KUKA KRL program: MyProgram_188().src

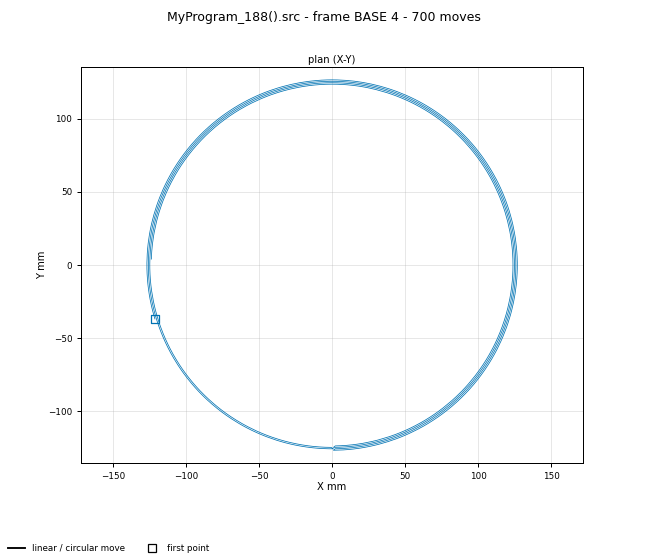
[picture p0: tool path of MyProgram_188().src in frame BASE 4, 700 of 700 moves have a stored position in this frame; points joined in program order, loops and branches not executed]
&ACCESS RVP
&REL 1
&PARAM TEMPLATE = C:\KRC\Roboter\Template\vorgabe
&PARAM EDITMASK = *
DEF MyProgram_188()
; ---- Setting reference (Base) ----
$BASE = BASE_DATA[4]

; --------------------------
; ---- Setting tool (TCP) ----
$TOOL = TOOL_DATA[3]
; --------------------------

$VEL.CP = VEL_APROX_PRINT
Startdeposition()
$VEL.CP = VEL_PRINT
LIN {X -121.2138,Y -36.8642,Z 137,A -166.8742,B 24.9598,C -1.4645,E1 24.8465,E2 613.2889} C_DIS
LIN {X -122.0831,Y -33.8748,Z 137,A -168.3082,B 24.9596,C -1.4677,E1 24.8454,E2 614.7236} C_DIS
LIN {X -122.8265,Y -31.0709,Z 137,A -169.6455,B 24.9595,C -1.4706,E1 24.8445,E2 616.0617} C_DIS
LIN {X -123.5708,Y -27.965,Z 137,A -171.133,B 24.9593,C -1.4732,E1 24.8435,E2 617.5517} C_DIS
LIN {X -124.4803,Y -23.589,Z 137,A -173.1147,B 24.9589,C -1.4814,E1 24.8424,E2 619.5256} C_DIS
LIN {X -125.0881,Y -20.1308,Z 137,A -174.7108,B 24.9586,C -1.4861,E1 24.8417,E2 621.1201} C_DIS
LIN {X -125.6254,Y -16.433,Z 137,A -176.4459,B 24.9584,C -1.4895,E1 24.841,E2 622.8573} C_DIS
LIN {X -126.0094,Y -13.1745,Z 137,A -177.8897,B 24.9581,C -1.4961,E1 24.8406,E2 624.2941} C_DIS
LIN {X -126.3219,Y -9.7379,Z 137,A -179.5918,B 24.9581,C -1.4948,E1 24.8402,E2 626.0096} C_DIS
LIN {X -126.5479,Y -6.1219,Z 137,A 178.8842,B 24.9575,C -1.5053,E1 24.8399,E2 627.5177} C_DIS
LIN {X -126.67,Y -2.6015,Z 137,A 177.1602,B 24.9575,C -1.5046,E1 24.8399,E2 629.2537} C_DIS
LIN {X -126.6899,Y 1.403,Z 137,A 175.4591,B 24.957,C -1.5155,E1 24.8399,E2 630.9392} C_DIS
LIN {X -126.5902,Y 5.1764,Z 137,A 173.7113,B 24.9568,C -1.5193,E1 24.8399,E2 632.6884} C_DIS
LIN {X -126.4456,Y 7.9589,Z 137,A 172.4536,B 24.9565,C -1.5235,E1 24.8402,E2 633.9435} C_DIS
LIN {X -126.1864,Y 11.3702,Z 137,A 170.907,B 24.9562,C -1.5286,E1 24.8405,E2 635.4873} C_DIS
LIN {X -125.7902,Y 15.1199,Z 137,A 169.1622,B 24.956,C -1.5325,E1 24.8411,E2 637.2334} C_DIS
LIN {X -125.3864,Y 18.1682,Z 137,A 167.7803,B 24.9557,C -1.5374,E1 24.8416,E2 638.6117} C_DIS
LIN {X -124.9317,Y 21.0685,Z 137,A 166.3962,B 24.9557,C -1.5392,E1 24.8422,E2 639.9998} C_DIS
LIN {X -124.3869,Y 24.0779,Z 137,A 165.0026,B 24.9554,C -1.5433,E1 24.8429,E2 641.392} C_DIS
LIN {X -123.5065,Y 28.2467,Z 137,A 163.0731,B 24.955,C -1.5494,E1 24.8441,E2 643.3182} C_DIS
LIN {X -122.739,Y 31.4153,Z 137,A 161.63,B 24.9547,C -1.5556,E1 24.845,E2 644.7551} C_DIS
LIN {X -121.9722,Y 34.2715,Z 137,A 160.2417,B 24.9545,C -1.5576,E1 24.8461,E2 646.1466} C_DIS
LIN {X -120.9226,Y 37.8158,Z 137,A 158.5823,B 24.9542,C -1.5635,E1 24.8474,E2 647.8016} C_DIS
LIN {X -120.1284,Y 40.2607,Z 137,A 157.4077,B 24.954,C -1.5666,E1 24.8484,E2 648.9753} C_DIS
LIN {X -119.0964,Y 43.2181,Z 137,A 155.982,B 24.9538,C -1.5707,E1 24.8498,E2 650.3994} C_DIS
LIN {X -117.9044,Y 46.3735,Z 137,A 154.4616,B 24.9535,C -1.5757,E1 24.8513,E2 651.9164} C_DIS
LIN {X -116.6051,Y 49.5537,Z 137,A 152.8791,B 24.9533,C -1.5792,E1 24.853,E2 653.4993} C_DIS
LIN {X -115.5382,Y 51.9875,Z 137,A 151.6701,B 24.9531,C -1.5826,E1 24.8543,E2 654.7069} C_DIS
LIN {X -114.1439,Y 54.9818,Z 137,A 150.1755,B 24.9528,C -1.5871,E1 24.8561,E2 656.1989} C_DIS
LIN {X -112.5436,Y 58.1916,Z 137,A 148.4062,B 24.9529,C -1.5853,E1 24.8584,E2 657.9819} C_DIS
LIN {X -110.5519,Y 61.8908,Z 137,A 146.5051,B 24.9526,C -1.591,E1 24.8609,E2 659.8796} C_DIS
LIN {X -108.3456,Y 65.6764,Z 137,A 144.5451,B 24.9522,C -1.5977,E1 24.8637,E2 661.8337} C_DIS
LIN {X -106.0689,Y 69.2941,Z 137,A 142.5626,B 24.952,C -1.601,E1 24.8667,E2 663.8183} C_DIS
LIN {X -103.768,Y 72.6946,Z 137,A 140.68,B 24.9517,C -1.6051,E1 24.8697,E2 665.7005} C_DIS
LIN {X -101.3771,Y 75.9934,Z 137,A 138.8143,B 24.9515,C -1.6091,E1 24.8728,E2 667.5656} C_DIS
LIN {X -98.705,Y 79.4322,Z 137,A 136.8715,B 24.9511,C -1.6156,E1 24.8761,E2 669.5021} C_DIS
LIN {X -95.9842,Y 82.6994,Z 137,A 134.9801,B 24.9507,C -1.6221,E1 24.8795,E2 671.3866} C_DIS
LIN {X -93.1998,Y 85.8252,Z 137,A 133.087,B 24.9504,C -1.627,E1 24.8831,E2 673.2766} C_DIS
LIN {X -90.3574,Y 88.8127,Z 137,A 131.2166,B 24.9501,C -1.6314,E1 24.8867,E2 675.1446} C_DIS
LIN {X -87.5001,Y 91.629,Z 137,A 129.3359,B 24.9501,C -1.6328,E1 24.8905,E2 677.0299} C_DIS
LIN {X -84.2229,Y 94.651,Z 137,A 127.3353,B 24.9497,C -1.6382,E1 24.8946,E2 679.0256} C_DIS
LIN {X -81.1209,Y 97.3227,Z 137,A 125.4906,B 24.9494,C -1.6427,E1 24.8985,E2 680.8666} C_DIS
LIN {X -77.9388,Y 99.8892,Z 137,A 123.5646,B 24.9494,C -1.6432,E1 24.9027,E2 682.7985} C_DIS
LIN {X -74.6821,Y 102.3469,Z 137,A 121.7215,B 24.9492,C -1.6472,E1 24.9069,E2 684.6387} C_DIS
LIN {X -71.2136,Y 104.7894,Z 137,A 119.7906,B 24.9489,C -1.6506,E1 24.9113,E2 686.5683} C_DIS
LIN {X -67.4012,Y 107.2814,Z 137,A 117.7556,B 24.9486,C -1.6557,E1 24.9161,E2 688.5976} C_DIS
LIN {X -63.8253,Y 109.447,Z 137,A 115.8771,B 24.9484,C -1.6597,E1 24.9206,E2 690.4722} C_DIS
LIN {X -60.3177,Y 111.4185,Z 137,A 113.9755,B 24.9484,C -1.6591,E1 24.9252,E2 692.3807} C_DIS
LIN {X -57.2259,Y 113.0352,Z 137,A 112.5422,B 24.9478,C -1.6685,E1 24.9287,E2 693.7956} C_DIS
LIN {X -54.374,Y 114.4343,Z 137,A 111.0509,B 24.9478,C -1.6683,E1 24.9325,E2 695.2913} C_DIS
LIN {X -51.4868,Y 115.7621,Z 137,A 109.6321,B 24.9477,C -1.6713,E1 24.9361,E2 696.7063} C_DIS
LIN {X -48.5808,Y 117.0114,Z 137,A 108.2322,B 24.9474,C -1.6748,E1 24.9397,E2 698.1011} C_DIS
LIN {X -45.6781,Y 118.1747,Z 137,A 106.753,B 24.9475,C -1.6738,E1 24.9436,E2 699.5861} C_DIS
LIN {X -42.385,Y 119.3968,Z 137,A 105.2355,B 24.9472,C -1.6791,E1 24.9475,E2 701.0938} C_DIS
LIN {X -39.5637,Y 120.3606,Z 137,A 103.8984,B 24.947,C -1.6813,E1 24.951,E2 702.4283} C_DIS
LIN {X -36.8296,Y 121.2244,Z 137,A 102.5937,B 24.947,C -1.6825,E1 24.9545,E2 703.7325} C_DIS
LIN {X -33.9371,Y 122.0657,Z 137,A 101.2091,B 24.947,C -1.6829,E1 24.9582,E2 705.1184} C_DIS
LIN {X -30.7333,Y 122.9121,Z 137,A 99.7525,B 24.9467,C -1.6864,E1 24.9622,E2 706.5687} C_DIS
LIN {X -27.965,Y 123.5709,Z 137,A 98.428,B 24.9467,C -1.6858,E1 24.9658,E2 707.8964} C_DIS
LIN {X -25.2359,Y 124.1567,Z 137,A 97.1229,B 24.9468,C -1.6849,E1 24.9694,E2 709.2052} C_DIS
LIN {X -22.0763,Y 124.7576,Z 137,A 95.6519,B 24.9468,C -1.6852,E1 24.9734,E2 710.677} C_DIS
LIN {X -18.7911,Y 125.2957,Z 137,A 94.2196,B 24.9465,C -1.6898,E1 24.9773,E2 712.0998} C_DIS
LIN {X -16.384,Y 125.6318,Z 137,A 93.0717,B 24.9465,C -1.6881,E1 24.9805,E2 713.2524} C_DIS
LIN {X -12.9917,Y 126.029,Z 137,A 91.5793,B 24.9464,C -1.6915,E1 24.9846,E2 714.7379} C_DIS
LIN {X -10.516,Y 126.2586,Z 137,A 90.4426,B 24.9464,C -1.6915,E1 24.9878,E2 715.8751} C_DIS
LIN {X -7.235,Y 126.4902,Z 137,A 88.7929,B 24.9468,C -1.6843,E1 24.9924,E2 717.5425} C_DIS
LIN {X -3.5172,Y 126.6469,Z 137,A 87.2244,B 24.9465,C -1.6903,E1 24.9968,E2 719.0969} C_DIS
LIN {X -0.2731,Y 126.6962,Z 137,A 85.6356,B 24.9468,C -1.6848,E1 25.0013,E2 720.6988} C_DIS
LIN {X 3.5292,Y 126.6466,Z 137,A 84.035,B 24.9464,C -1.6907,E1 25.0057,E2 722.285} C_DIS
LIN {X 6.7282,Y 126.5175,Z 137,A 82.6482,B 24.9462,C -1.6937,E1 25.0095,E2 723.6643} C_DIS
LIN {X 9.3313,Y 126.3516,Z 137,A 81.3748,B 24.9465,C -1.6892,E1 25.0131,E2 724.9479} C_DIS
LIN {X 12.3501,Y 126.0925,Z 137,A 80.0692,B 24.9463,C -1.6921,E1 25.0167,E2 726.2457} C_DIS
LIN {X 15.1123,Y 125.7911,Z 137,A 78.7888,B 24.9464,C -1.6908,E1 25.0203,E2 727.5284} C_DIS
LIN {X 18.1682,Y 125.3864,Z 137,A 77.4376,B 24.9464,C -1.6925,E1 25.024,E2 728.8744} C_DIS
LIN {X 21.0976,Y 124.9268,Z 137,A 76.0462,B 24.9465,C -1.6896,E1 25.0279,E2 730.2713} C_DIS
LIN {X 24.0358,Y 124.3949,Z 137,A 74.7449,B 24.9464,C -1.6914,E1 25.0314,E2 731.5668} C_DIS
LIN {X 26.9849,Y 123.7886,Z 137,A 73.3155,B 24.9466,C -1.6875,E1 25.0353,E2 733.0037} C_DIS
LIN {X 29.8689,Y 123.1244,Z 137,A 72.0099,B 24.9466,C -1.6883,E1 25.0389,E2 734.3055} C_DIS
LIN {X 32.8933,Y 122.3512,Z 137,A 70.5572,B 24.9468,C -1.6854,E1 25.0428,E2 735.7628} C_DIS
LIN {X 36.301,Y 121.3857,Z 137,A 69.0155,B 24.9467,C -1.6871,E1 25.0469,E2 737.2978} C_DIS
LIN {X 38.8012,Y 120.6078,Z 137,A 67.8234,B 24.9467,C -1.6858,E1 25.0501,E2 738.4908} C_DIS
LIN {X 41.7479,Y 119.6198,Z 137,A 66.4186,B 24.9468,C -1.6846,E1 25.0538,E2 739.8957} C_DIS
LIN {X 44.6859,Y 118.5535,Z 137,A 64.9566,B 24.9471,C -1.6809,E1 25.0577,E2 741.3634} C_DIS
LIN {X 47.7378,Y 117.3582,Z 137,A 63.4947,B 24.9471,C -1.6804,E1 25.0614,E2 742.8233} C_DIS
LIN {X 50.5237,Y 116.1857,Z 137,A 62.166,B 24.9471,C -1.6807,E1 25.0648,E2 744.1479} C_DIS
LIN {X 53.4175,Y 114.8839,Z 137,A 60.7112,B 24.9472,C -1.678,E1 25.0685,E2 745.6054} C_DIS
LIN {X 56.7659,Y 113.2693,Z 137,A 59.0497,B 24.9473,C -1.6768,E1 25.0727,E2 747.2653} C_DIS
LIN {X 60.0362,Y 111.5698,Z 137,A 57.3378,B 24.9476,C -1.6723,E1 25.0769,E2 748.983} C_DIS
LIN {X 63.3593,Y 109.7168,Z 137,A 55.5741,B 24.9479,C -1.6677,E1 25.0812,E2 750.7524} C_DIS
LIN {X 66.8236,Y 107.6419,Z 137,A 53.7522,B 24.948,C -1.6651,E1 25.0856,E2 752.5748} C_DIS
LIN {X 70.253,Y 105.4356,Z 137,A 51.9188,B 24.9482,C -1.6626,E1 25.0899,E2 754.408} C_DIS
LIN {X 73.8234,Y 102.9674,Z 137,A 49.9585,B 24.9484,C -1.6594,E1 25.0944,E2 756.3691} C_DIS
LIN {X 77.2932,Y 100.3896,Z 137,A 47.9978,B 24.9486,C -1.6555,E1 25.0987,E2 758.3319} C_DIS
LIN {X 80.5773,Y 97.7729,Z 137,A 46.0862,B 24.9489,C -1.6513,E1 25.1029,E2 760.2464} C_DIS
LIN {X 83.813,Y 95.0134,Z 137,A 44.2,B 24.949,C -1.6493,E1 25.1069,E2 762.1298} C_DIS
LIN {X 87.0418,Y 92.0645,Z 137,A 42.2885,B 24.949,C -1.6485,E1 25.1108,E2 764.0354} C_DIS
LIN {X 89.8701,Y 89.3057,Z 137,A 40.4805,B 24.9494,C -1.6436,E1 25.1144,E2 765.8474} C_DIS
LIN {X 92.603,Y 86.4688,Z 137,A 38.6715,B 24.9497,C -1.6382,E1 25.1178,E2 767.6613} C_DIS
LIN {X 95.5433,Y 83.2084,Z 137,A 36.7072,B 24.9499,C -1.6346,E1 25.1215,E2 769.6251} C_DIS
LIN {X 98.3622,Y 79.8573,Z 137,A 34.7605,B 24.9501,C -1.6316,E1 25.1249,E2 771.5701} C_DIS
LIN {X 100.8855,Y 76.6448,Z 137,A 32.8699,B 24.9505,C -1.6248,E1 25.1282,E2 773.4678} C_DIS
LIN {X 103.4105,Y 73.2015,Z 137,A 30.9602,B 24.9508,C -1.621,E1 25.1313,E2 775.3773} C_DIS
LIN {X 105.7474,Y 69.783,Z 137,A 29.1171,B 24.951,C -1.6176,E1 25.1342,E2 777.2192} C_DIS
LIN {X 108.0663,Y 66.135,Z 137,A 27.1864,B 24.9512,C -1.6136,E1 25.137,E2 779.1495} C_DIS
LIN {X 110.25,Y 62.428,Z 137,A 25.1881,B 24.9517,C -1.6055,E1 25.1398,E2 781.1565} C_DIS
LIN {X 112.2765,Y 58.7001,Z 137,A 23.4009,B 24.9517,C -1.607,E1 25.1422,E2 782.9309} C_DIS
LIN {X 113.7411,Y 55.8096,Z 137,A 21.976,B 24.9517,C -1.6049,E1 25.1439,E2 784.3531} C_DIS
LIN {X 115.1253,Y 52.8956,Z 137,A 20.5325,B 24.9519,C -1.6015,E1 25.1456,E2 785.7969} C_DIS
LIN {X 116.4302,Y 49.9581,Z 137,A 19.1101,B 24.9521,C -1.5988,E1 25.1472,E2 787.2178} C_DIS
LIN {X 117.6066,Y 47.1217,Z 137,A 17.7058,B 24.9524,C -1.5939,E1 25.1487,E2 788.6259} C_DIS
LIN {X 118.8554,Y 43.8799,Z 137,A 16.1423,B 24.9527,C -1.5896,E1 25.1503,E2 790.191} C_DIS
LIN {X 119.9606,Y 40.7648,Z 137,A 14.6629,B 24.9529,C -1.5858,E1 25.1516,E2 791.6709} C_DIS
LIN {X 121.2244,Y 36.8296,Z 137,A 12.8239,B 24.9531,C -1.5817,E1 25.1532,E2 793.5092} C_DIS
LIN {X 122.0831,Y 33.8748,Z 137,A 11.419,B 24.9534,C -1.5766,E1 25.1542,E2 794.9179} C_DIS
LIN {X 122.7978,Y 31.1838,Z 137,A 10.1656,B 24.9536,C -1.573,E1 25.1551,E2 796.1727} C_DIS
LIN {X 123.5567,Y 28.027,Z 137,A 8.6985,B 24.9539,C -1.5684,E1 25.1561,E2 797.642} C_DIS
LIN {X 124.2016,Y 25.0154,Z 137,A 7.3417,B 24.9541,C -1.5659,E1 25.1568,E2 798.9969} C_DIS
LIN {X 124.7582,Y 22.0728,Z 137,A 5.9489,B 24.9544,C -1.5596,E1 25.1575,E2 800.3965} C_DIS
LIN {X 125.3864,Y 18.1682,Z 137,A 4.1663,B 24.9547,C -1.5541,E1 25.1583,E2 802.1814} C_DIS
LIN {X 125.8327,Y 14.7633,Z 137,A 2.6629,B 24.9549,C -1.5517,E1 25.1588,E2 803.6817} C_DIS
LIN {X 126.1447,Y 11.8066,Z 137,A 1.3757,B 24.9549,C -1.5503,E1 25.1592,E2 804.9645} C_DIS
LIN {X 126.3534,Y 9.3065,Z 137,A 0.169,B 24.9554,C -1.5428,E1 25.1594,E2 806.1817} C_DIS
LIN {X 126.5718,Y 5.6482,Z 137,A -1.5786,B 24.956,C -1.5326,E1 25.1597,E2 807.9429} C_DIS
LIN {X 126.6822,Y 1.871,Z 137,A -3.0955,B 24.9557,C -1.5371,E1 25.1597,E2 809.4402} C_DIS
LIN {X 126.675,Y -2.303,Z 137,A -4.9812,B 24.9561,C -1.531,E1 25.1597,E2 811.3291} C_DIS
LIN {X 126.5718,Y -5.6482,Z 137,A -6.6352,B 24.9568,C -1.5186,E1 25.1596,E2 813.0024} C_DIS
LIN {X 126.3525,Y -9.3195,Z 137,A -8.2229,B 24.9568,C -1.5171,E1 25.1593,E2 814.5843} C_DIS
LIN {X 125.9422,Y -13.7988,Z 137,A -10.1568,B 24.957,C -1.5157,E1 25.1587,E2 816.5101} C_DIS
LIN {X 125.6134,Y -16.5243,Z 137,A -11.4361,B 24.9573,C -1.5096,E1 25.1583,E2 817.7961} C_DIS
LIN {X 125.1656,Y -19.6315,Z 137,A -12.8094,B 24.9574,C -1.5074,E1 25.1577,E2 819.1666} C_DIS
LIN {X 124.5973,Y -22.9721,Z 137,A -14.3281,B 24.9577,C -1.503,E1 25.157,E2 820.6867} C_DIS
LIN {X 124.1301,Y -25.3669,Z 137,A -15.4629,B 24.958,C -1.4978,E1 25.1564,E2 821.8272} C_DIS
LIN {X 123.4519,Y -28.4859,Z 137,A -16.8624,B 24.9581,C -1.4954,E1 25.1555,E2 823.2241} C_DIS
LIN {X 122.7808,Y -31.251,Z 137,A -18.1828,B 24.9584,C -1.4895,E1 25.1546,E2 824.5509} C_DIS
LIN {X 121.9542,Y -34.3358,Z 137,A -19.6462,B 24.9588,C -1.4838,E1 25.1535,E2 826.0192} C_DIS
LIN {X 121.0458,Y -37.4134,Z 137,A -21.0246,B 24.9588,C -1.4829,E1 25.1524,E2 827.3918} C_DIS
LIN {X 120.1236,Y -40.2754,Z 137,A -22.3706,B 24.959,C -1.4793,E1 25.1513,E2 828.7387} C_DIS
LIN {X 119.0964,Y -43.2181,Z 137,A -23.7896,B 24.9593,C -1.4743,E1 25.1499,E2 830.1615} C_DIS
LIN {X 117.959,Y -46.233,Z 137,A -25.2628,B 24.9596,C -1.4689,E1 25.1484,E2 831.6393} C_DIS
LIN {X 116.8498,Y -48.9678,Z 137,A -26.5831,B 24.9598,C -1.4655,E1 25.147,E2 832.9603} C_DIS
LIN {X 115.5296,Y -52.0066,Z 137,A -28.0516,B 24.9599,C -1.4624,E1 25.1454,E2 834.4281} C_DIS
LIN {X 114.0697,Y -55.1372,Z 137,A -29.5808,B 24.9601,C -1.4593,E1 25.1436,E2 835.9565} C_DIS
LIN {X 112.7846,Y -57.7181,Z 137,A -30.9081,B 24.9604,C -1.4541,E1 25.1419,E2 837.2888} C_DIS
LIN {X 111.0466,Y -60.9995,Z 137,A -32.7013,B 24.961,C -1.4431,E1 25.1395,E2 839.0986} C_DIS
LIN {X 109.0383,Y -64.5209,Z 137,A -34.5459,B 24.9613,C -1.4371,E1 25.1369,E2 840.9478} C_DIS
LIN {X 106.7947,Y -68.1694,Z 137,A -36.4283,B 24.9615,C -1.4343,E1 25.1341,E2 842.8273} C_DIS
LIN {X 104.54,Y -71.579,Z 137,A -38.2602,B 24.9617,C -1.4299,E1 25.1312,E2 844.6606} C_DIS
LIN {X 101.991,Y -75.1666,Z 137,A -40.2434,B 24.962,C -1.4247,E1 25.128,E2 846.6465} C_DIS
LIN {X 99.3845,Y -78.5813,Z 137,A -42.1465,B 24.9622,C -1.4214,E1 25.1247,E2 848.5482} C_DIS
LIN {X 96.7967,Y -81.7478,Z 137,A -44.0394,B 24.9625,C -1.4142,E1 25.1213,E2 850.4495} C_DIS
LIN {X 93.9933,Y -84.9556,Z 137,A -45.9542,B 24.9628,C -1.4098,E1 25.1178,E2 852.366} C_DIS
LIN {X 91.1218,Y -88.0282,Z 137,A -47.8202,B 24.9629,C -1.4068,E1 25.1142,E2 854.2311} C_DIS
LIN {X 88.2296,Y -90.9269,Z 137,A -49.6636,B 24.9631,C -1.4027,E1 25.1105,E2 856.0765} C_DIS
LIN {X 85.0393,Y -93.9174,Z 137,A -51.5733,B 24.9632,C -1.4014,E1 25.1066,E2 857.9814} C_DIS
LIN {X 81.9619,Y -96.6147,Z 137,A -53.4151,B 24.9634,C -1.3976,E1 25.1027,E2 859.8251} C_DIS
LIN {X 79.0085,Y -99.0445,Z 137,A -55.1915,B 24.9637,C -1.3913,E1 25.0989,E2 861.6095} C_DIS
LIN {X 75.5578,Y -101.7014,Z 137,A -57.0941,B 24.9637,C -1.3904,E1 25.0946,E2 863.5073} C_DIS
LIN {X 72.6054,Y -103.8301,Z 137,A -58.8282,B 24.9642,C -1.3825,E1 25.0907,E2 865.2541} C_DIS
LIN {X 69.1043,Y -106.1921,Z 137,A -60.6892,B 24.9642,C -1.3812,E1 25.0863,E2 867.1121} C_DIS
LIN {X 65.6764,Y -108.3456,Z 137,A -62.5109,B 24.9644,C -1.3781,E1 25.082,E2 868.9353} C_DIS
LIN {X 62.3043,Y -110.3195,Z 137,A -64.2998,B 24.9647,C -1.3737,E1 25.0777,E2 870.7291} C_DIS
LIN {X 58.3013,Y -112.4859,Z 137,A -66.2074,B 24.9644,C -1.3778,E1 25.073,E2 872.6217} C_DIS
LIN {X 55.8174,Y -113.7372,Z 137,A -67.4768,B 24.9646,C -1.3751,E1 25.0698,E2 873.894} C_DIS
LIN {X 53.0118,Y -115.0716,Z 137,A -68.8875,B 24.9647,C -1.3726,E1 25.0662,E2 875.307} C_DIS
LIN {X 50.1185,Y -116.3609,Z 137,A -70.3142,B 24.9648,C -1.3707,E1 25.0626,E2 876.7348} C_DIS
LIN {X 47.1217,Y -117.6066,Z 137,A -71.7607,B 24.9648,C -1.3696,E1 25.0588,E2 878.1806} C_DIS
LIN {X 43.9852,Y -118.816,Z 137,A -73.2535,B 24.9649,C -1.3689,E1 25.0549,E2 879.6718} C_DIS
LIN {X 41.0279,Y -119.8694,Z 137,A -74.6654,B 24.9649,C -1.3674,E1 25.0512,E2 881.0844} C_DIS
LIN {X 38.1452,Y -120.8174,Z 137,A -76.0333,B 24.9651,C -1.3659,E1 25.0476,E2 882.4532} C_DIS
LIN {X 35.3525,Y -121.6634,Z 137,A -77.3694,B 24.9651,C -1.3636,E1 25.044,E2 883.7925} C_DIS
LIN {X 32.2785,Y -122.5152,Z 137,A -78.8083,B 24.9652,C -1.3622,E1 25.0401,E2 885.2324} C_DIS
LIN {X 29.1154,Y -123.306,Z 137,A -80.259,B 24.9652,C -1.3619,E1 25.0362,E2 886.6817} C_DIS
LIN {X 25.9996,Y -124.0013,Z 137,A -81.7173,B 24.9654,C -1.3598,E1 25.0322,E2 888.1431} C_DIS
LIN {X 22.0728,Y -124.7582,Z 137,A -83.5692,B 24.9655,C -1.3562,E1 25.0271,E2 890.0014} C_DIS
LIN {X 18.6854,Y -125.3121,Z 137,A -85.0617,B 24.9655,C -1.358,E1 25.023,E2 891.4883} C_DIS
LIN {X 14.2804,Y -125.8904,Z 137,A -87.216,B 24.9659,C -1.3495,E1 25.017,E2 893.661} C_DIS
LIN {X 10.7424,Y -126.2394,Z 137,A -88.6882,B 24.9656,C -1.3554,E1 25.0129,E2 895.1184} C_DIS
LIN {X 7.55,Y -126.4708,Z 137,A -90.1637,B 24.9656,C -1.3533,E1 25.0088,E2 896.5981} C_DIS
LIN {X 3.5794,Y -126.6452,Z 137,A -91.962,B 24.9657,C -1.3526,E1 25.0038,E2 898.3975} C_DIS
LIN {X 0.8999,Y -126.6905,Z 137,A -92.7577,B 24.9647,C -1.3729,E1 25.0017,E2 899.145} C_DIS
Enddeposition()
LIN {X 0.8999,Y -126.6905,Z 137,A -92.7577,B 24.9647,C -1.3729,E1 25.0017,E2 899.145} C_DIS
Startdeposition()
$VEL.CP = VEL_PRINT
LIN {X 2.0498,Y -125.6939,Z 137,A -91.9702,B 24.9631,C -1.4033,E1 25.0041,E2 898.2858} C_DIS
LIN {X 6.1944,Y -125.5579,Z 137,A -90.1113,B 24.9631,C -1.4024,E1 25.0093,E2 896.4294} C_DIS
LIN {X 9.9563,Y -125.3171,Z 137,A -88.2949,B 24.9629,C -1.4081,E1 25.0144,E2 894.6004} C_DIS
LIN {X 13.8589,Y -124.9448,Z 137,A -86.5088,B 24.9629,C -1.4091,E1 25.0193,E2 892.8131} C_DIS
LIN {X 17.8799,Y -124.4324,Z 137,A -84.7165,B 24.9629,C -1.4076,E1 25.0243,E2 891.0259} C_DIS
LIN {X 22.0203,Y -123.7667,Z 137,A -82.5492,B 24.9621,C -1.4219,E1 25.0303,E2 888.8269} C_DIS
LIN {X 26.8174,Y -122.8169,Z 137,A -80.5783,B 24.9627,C -1.4109,E1 25.0356,E2 886.8846} C_DIS
LIN {X 30.7223,Y -121.8985,Z 137,A -78.7593,B 24.9627,C -1.4123,E1 25.0406,E2 885.0649} C_DIS
LIN {X 36.9269,Y -120.1643,Z 137,A -75.8722,B 24.9626,C -1.4131,E1 25.0483,E2 882.1807} C_DIS
LIN {X 40.5195,Y -119.0029,Z 137,A -73.625,B 24.961,C -1.442,E1 25.0544,E2 879.8696} C_DIS
LIN {X 44.5267,Y -117.5611,Z 137,A -72.145,B 24.9622,C -1.4212,E1 25.0582,E2 878.4419} C_DIS
LIN {X 48.4066,Y -116.0165,Z 137,A -70.3276,B 24.9622,C -1.4196,E1 25.0628,E2 876.6325} C_DIS
LIN {X 51.4937,Y -114.6798,Z 137,A -68.8482,B 24.9622,C -1.4192,E1 25.0666,E2 875.1577} C_DIS
LIN {X 54.2622,Y -113.3959,Z 137,A -67.41,B 24.962,C -1.4239,E1 25.0703,E2 873.7121} C_DIS
LIN {X 57.2555,Y -111.9146,Z 137,A -65.8413,B 24.9618,C -1.4288,E1 25.0742,E2 872.136} C_DIS
LIN {X 61.0429,Y -109.8966,Z 137,A -63.8208,B 24.9614,C -1.4356,E1 25.0792,E2 870.1054} C_DIS
LIN {X 64.6843,Y -107.794,Z 137,A -61.9156,B 24.9612,C -1.4386,E1 25.0838,E2 868.1989} C_DIS
LIN {X 68.8957,Y -105.1519,Z 137,A -59.6159,B 24.9609,C -1.4448,E1 25.0892,E2 865.892} C_DIS
LIN {X 72.2281,Y -102.8915,Z 137,A -58.0605,B 24.9615,C -1.4342,E1 25.0927,E2 864.367} C_DIS
LIN {X 74.819,Y -101.0233,Z 137,A -56.4177,B 24.9608,C -1.4469,E1 25.0964,E2 862.7001} C_DIS
LIN {X 79.728,Y -97.1955,Z 137,A -52.9744,B 24.9587,C -1.4847,E1 25.1041,E2 859.1804} C_DIS
LIN {X 83.6631,Y -93.8298,Z 137,A -51.4878,B 24.9609,C -1.4448,E1 25.107,E2 857.7937} C_DIS
LIN {X 88.4403,Y -89.3411,Z 137,A -48.5068,B 24.9605,C -1.4517,E1 25.1131,E2 854.809} C_DIS
LIN {X 92.666,Y -84.95,Z 137,A -45.7554,B 24.9602,C -1.4573,E1 25.1184,E2 852.0562} C_DIS
LIN {X 97.3178,Y -79.5784,Z 137,A -41.9157,B 24.958,C -1.4972,E1 25.1255,E2 848.1399} C_DIS
LIN {X 99.7776,Y -76.4717,Z 137,A -40.637,B 24.9593,C -1.4745,E1 25.1275,E2 846.9207} C_DIS
LIN {X 102.0052,Y -73.4749,Z 137,A -38.7782,B 24.9586,C -1.4874,E1 25.1306,E2 845.0404} C_DIS
LIN {X 104.4909,Y -69.8938,Z 137,A -36.8094,B 24.9583,C -1.4922,E1 25.1337,E2 843.0701} C_DIS
LIN {X 106.7509,Y -66.3906,Z 137,A -34.9407,B 24.9581,C -1.496,E1 25.1365,E2 841.2017} C_DIS
LIN {X 108.9996,Y -62.6317,Z 137,A -33.2076,B 24.9585,C -1.4882,E1 25.1389,E2 839.4961} C_DIS
LIN {X 110.5013,Y -59.9419,Z 137,A -31.5166,B 24.9574,C -1.5074,E1 25.1413,E2 837.7687} C_DIS
LIN {X 112.555,Y -55.9871,Z 137,A -29.5489,B 24.9573,C -1.5102,E1 25.1437,E2 835.8047} C_DIS
LIN {X 114.2588,Y -52.4222,Z 137,A -27.86,B 24.9573,C -1.5099,E1 25.1457,E2 834.1257} C_DIS
LIN {X 115.7184,Y -49.1203,Z 137,A -26.0235,B 24.9564,C -1.525,E1 25.1478,E2 832.2636} C_DIS
LIN {X 117.2618,Y -45.3073,Z 137,A -24.3022,B 24.9566,C -1.5229,E1 25.1495,E2 830.5568} C_DIS
LIN {X 119.3041,Y -39.6178,Z 137,A -21.9887,B 24.9574,C -1.5085,E1 25.1517,E2 828.2902} C_DIS
LIN {X 120.6701,Y -35.2389,Z 137,A -19.5925,B 24.9561,C -1.5311,E1 25.1537,E2 825.8543} C_DIS
LIN {X 121.4981,Y -32.2688,Z 137,A -18.1367,B 24.9557,C -1.5383,E1 25.1547,E2 824.39} C_DIS
LIN {X 122.6925,Y -27.3862,Z 137,A -15.9152,B 24.9554,C -1.5421,E1 25.1562,E2 822.1725} C_DIS
LIN {X 123.2933,Y -24.5385,Z 137,A -14.4918,B 24.9549,C -1.5515,E1 25.157,E2 820.7351} C_DIS
LIN {X 123.9877,Y -20.7397,Z 137,A -12.7869,B 24.9547,C -1.5544,E1 25.1578,E2 819.0335} C_DIS
LIN {X 124.5514,Y -17.0459,Z 137,A -10.9741,B 24.9541,C -1.5657,E1 25.1585,E2 817.2046} C_DIS
LIN {X 125.0205,Y -13.1556,Z 137,A -9.3415,B 24.9541,C -1.5636,E1 25.159,E2 815.5867} C_DIS
LIN {X 125.3611,Y -9.3681,Z 137,A -7.5376,B 24.9536,C -1.573,E1 25.1594,E2 813.7713} C_DIS
LIN {X 125.607,Y -5.1052,Z 137,A -5.6603,B 24.9535,C -1.5758,E1 25.1597,E2 811.8986} C_DIS
LIN {X 125.7063,Y -1.1881,Z 137,A -3.8811,B 24.9531,C -1.5813,E1 25.1597,E2 810.117} C_DIS
LIN {X 125.6822,Y 2.7521,Z 137,A -1.9946,B 24.9525,C -1.5919,E1 25.1597,E2 808.2166} C_DIS
LIN {X 125.5349,Y 6.6501,Z 137,A -0.3058,B 24.9525,C -1.5931,E1 25.1595,E2 806.5352} C_DIS
LIN {X 125.2677,Y 10.5416,Z 137,A 1.441,B 24.9522,C -1.5973,E1 25.1591,E2 804.7888} C_DIS
LIN {X 124.8619,Y 14.5843,Z 137,A 3.2805,B 24.9519,C -1.6027,E1 25.1586,E2 802.9476} C_DIS
LIN {X 124.3998,Y 18.108,Z 137,A 4.9763,B 24.9513,C -1.6119,E1 25.1579,E2 801.2401} C_DIS
LIN {X 123.7536,Y 22.094,Z 137,A 6.6905,B 24.9513,C -1.6112,E1 25.1571,E2 799.5376} C_DIS
LIN {X 123.0618,Y 25.676,Z 137,A 8.5419,B 24.9504,C -1.6263,E1 25.1561,E2 797.6613} C_DIS
LIN {X 122.1388,Y 29.7536,Z 137,A 10.1871,B 24.9509,C -1.6187,E1 25.155,E2 796.0435} C_DIS
LIN {X 121.3302,Y 32.8986,Z 137,A 11.764,B 24.9503,C -1.6284,E1 25.1539,E2 794.4529} C_DIS
LIN {X 120.2502,Y 36.6465,Z 137,A 13.464,B 24.9503,C -1.6298,E1 25.1526,E2 792.7592} C_DIS
LIN {X 118.6868,Y 41.4314,Z 137,A 15.8288,B 24.9496,C -1.6405,E1 25.1504,E2 790.3827} C_DIS
LIN {X 117.2235,Y 45.406,Z 137,A 17.697,B 24.9494,C -1.643,E1 25.1486,E2 788.5188} C_DIS
LIN {X 115.899,Y 48.6878,Z 137,A 19.3009,B 24.9491,C -1.6473,E1 25.1469,E2 786.9136} C_DIS
LIN {X 114.2218,Y 52.5022,Z 137,A 22.3006,B 24.9452,C -1.7105,E1 25.1433,E2 783.7812} C_DIS
LIN {X 110.9544,Y 59.0985,Z 137,A 24.3603,B 24.9488,C -1.6522,E1 25.1408,E2 781.8699} C_DIS
LIN {X 109.189,Y 62.2996,Z 137,A 25.9661,B 24.9488,C -1.6537,E1 25.1386,E2 780.269} C_DIS
LIN {X 107.6909,Y 64.8553,Z 137,A 27.5805,B 24.9477,C -1.671,E1 25.1363,E2 778.622} C_DIS
LIN {X 105.5057,Y 68.3522,Z 137,A 29.4638,B 24.9473,C -1.6762,E1 25.1334,E2 776.7359} C_DIS
LIN {X 103.0789,Y 71.9601,Z 137,A 31.3856,B 24.9473,C -1.6782,E1 25.1304,E2 774.8188} C_DIS
LIN {X 100.544,Y 75.4618,Z 137,A 33.4001,B 24.9468,C -1.6855,E1 25.127,E2 772.7969} C_DIS
LIN {X 97.8909,Y 78.8723,Z 137,A 35.3377,B 24.9466,C -1.6887,E1 25.1237,E2 770.8608} C_DIS
LIN {X 95.1032,Y 82.2126,Z 137,A 37.321,B 24.9463,C -1.6934,E1 25.1201,E2 768.8754} C_DIS
LIN {X 92.398,Y 85.2416,Z 137,A 39.1883,B 24.9459,C -1.6985,E1 25.1166,E2 767.0044} C_DIS
LIN {X 89.3931,Y 88.388,Z 137,A 41.1518,B 24.9457,C -1.7019,E1 25.1128,E2 765.0413} C_DIS
LIN {X 86.3642,Y 91.3494,Z 137,A 43.0383,B 24.9457,C -1.7037,E1 25.109,E2 763.1583} C_DIS
LIN {X 83.3372,Y 94.1191,Z 137,A 44.8419,B 24.9456,C -1.7042,E1 25.1052,E2 761.3608} C_DIS
LIN {X 80.206,Y 96.8012,Z 137,A 46.7913,B 24.9451,C -1.7114,E1 25.1011,E2 759.4018} C_DIS
LIN {X 76.8485,Y 99.4878,Z 137,A 48.7603,B 24.9448,C -1.7156,E1 25.0967,E2 757.4304} C_DIS
LIN {X 73.3707,Y 102.0799,Z 137,A 50.6563,B 24.9448,C -1.715,E1 25.0925,E2 755.5425} C_DIS
LIN {X 70.0715,Y 104.3722,Z 137,A 52.5813,B 24.9444,C -1.7228,E1 25.088,E2 753.6056} C_DIS
LIN {X 66.1874,Y 106.8774,Z 137,A 55.8085,B 24.9404,C -1.783,E1 25.0801,E2 750.2461} C_DIS
LIN {X 59.3509,Y 110.8195,Z 137,A 57.8598,B 24.9452,C -1.71,E1 25.0755,E2 748.3735} C_DIS
LIN {X 56.2857,Y 112.4077,Z 137,A 59.6621,B 24.9443,C -1.7234,E1 25.0709,E2 746.5444} C_DIS
LIN {X 53.9638,Y 113.5385,Z 137,A 60.833,B 24.9443,C -1.7246,E1 25.068,E2 745.3737} C_DIS
LIN {X 51.1226,Y 114.8457,Z 137,A 62.3073,B 24.944,C -1.7287,E1 25.0642,E2 743.8934} C_DIS
LIN {X 47.8328,Y 116.2561,Z 137,A 64.083,B 24.9434,C -1.7376,E1 25.0596,E2 742.1007} C_DIS
LIN {X 44.1657,Y 117.6963,Z 137,A 65.7139,B 24.9438,C -1.7313,E1 25.0554,E2 740.4885} C_DIS
LIN {X 40.9949,Y 118.8381,Z 137,A 67.2669,B 24.9437,C -1.7335,E1 25.0513,E2 738.9334} C_DIS
LIN {X 37.1044,Y 120.11,Z 137,A 68.9179,B 24.9443,C -1.7244,E1 25.047,E2 737.3069} C_DIS
LIN {X 34.0435,Y 121.0129,Z 137,A 70.5825,B 24.9435,C -1.7358,E1 25.0424,E2 735.6181} C_DIS
LIN {X 30.6125,Y 121.9264,Z 137,A 72.2258,B 24.9434,C -1.7381,E1 25.038,E2 733.972} C_DIS
LIN {X 26.0821,Y 122.9756,Z 137,A 74.3425,B 24.9434,C -1.739,E1 25.0322,E2 731.8559} C_DIS
LIN {X 22.1894,Y 123.7365,Z 137,A 76.1385,B 24.9434,C -1.7392,E1 25.0273,E2 730.0616} C_DIS
LIN {X 18.0662,Y 124.4058,Z 137,A 78.0242,B 24.9434,C -1.7389,E1 25.0221,E2 728.1784} C_DIS
LIN {X 14.5698,Y 124.8636,Z 137,A 79.7115,B 24.9431,C -1.7431,E1 25.0174,E2 726.4824} C_DIS
LIN {X 10.5748,Y 125.2649,Z 137,A 81.4469,B 24.9433,C -1.7387,E1 25.0126,E2 724.7584} C_DIS
LIN {X 6.5578,Y 125.5396,Z 137,A 83.3193,B 24.9433,C -1.7405,E1 25.0074,E2 722.8824} C_DIS
LIN {X 2.718,Y 125.6827,Z 137,A 85.1526,B 24.943,C -1.7443,E1 25.0022,E2 721.0407} C_DIS
LIN {X -1.3707,Y 125.7049,Z 137,A 87.012,B 24.943,C -1.7437,E1 24.997,E2 719.1827} C_DIS
LIN {X -5.3226,Y 125.5985,Z 137,A 88.7941,B 24.9431,C -1.7422,E1 24.9921,E2 717.4038} C_DIS
LIN {X -9.3182,Y 125.3648,Z 137,A 90.5965,B 24.9432,C -1.7404,E1 24.987,E2 715.6051} C_DIS
LIN {X -13.3298,Y 125.0018,Z 137,A 92.3418,B 24.9436,C -1.7351,E1 24.9822,E2 713.8713} C_DIS
LIN {X -16.5677,Y 124.6141,Z 137,A 93.8345,B 24.9436,C -1.7345,E1 24.9781,E2 712.3789} C_DIS
LIN {X -20.2162,Y 124.0751,Z 137,A 95.5865,B 24.9435,C -1.7367,E1 24.9732,E2 710.6201} C_DIS
LIN {X -23.6013,Y 123.4749,Z 137,A 97.1879,B 24.9435,C -1.7372,E1 24.9688,E2 709.0161} C_DIS
LIN {X -32.8557,Y 121.3416,Z 137,A 100.8975,B 24.9456,C -1.7037,E1 24.959,E2 705.381} C_DIS
LIN {X -40.7265,Y 118.9312,Z 137,A 105.0527,B 24.9447,C -1.7182,E1 24.9478,E2 701.1842} C_DIS
LIN {X -44.4836,Y 117.5773,Z 137,A 107.1542,B 24.944,C -1.729,E1 24.9422,E2 699.0527} C_DIS
LIN {X -48.2852,Y 116.0672,Z 137,A 108.8893,B 24.9445,C -1.7203,E1 24.9377,E2 697.3344} C_DIS
LIN {X -53.5105,Y 113.755,Z 137,A 111.4742,B 24.9449,C -1.7154,E1 24.9312,E2 694.755} C_DIS
LIN {X -57.7416,Y 111.6671,Z 137,A 113.7895,B 24.9446,C -1.7195,E1 24.9253,E2 692.4237} C_DIS
LIN {X -63.024,Y 108.7725,Z 137,A 116.3377,B 24.9455,C -1.7055,E1 24.9192,E2 689.9015} C_DIS
LIN {X -66.113,Y 106.9237,Z 137,A 118.1967,B 24.945,C -1.7125,E1 24.9147,E2 688.02} C_DIS
LIN {X -69.8325,Y 104.5318,Z 137,A 120.1824,B 24.9454,C -1.7072,E1 24.9101,E2 686.0404} C_DIS
LIN {X -73.4068,Y 102.0541,Z 137,A 122.1949,B 24.9456,C -1.7045,E1 24.9055,E2 684.0274} C_DIS
LIN {X -76.8119,Y 99.5161,Z 137,A 124.1472,B 24.9458,C -1.7011,E1 24.9011,E2 682.076} C_DIS
LIN {X -80.4219,Y 96.6224,Z 137,A 126.1938,B 24.9462,C -1.6936,E1 24.8967,E2 680.0397} C_DIS
LIN {X -83.5307,Y 93.948,Z 137,A 128.1388,B 24.9463,C -1.6928,E1 24.8926,E2 678.089} C_DIS
LIN {X -86.6512,Y 91.0775,Z 137,A 130.0939,B 24.9465,C -1.6892,E1 24.8887,E2 676.1345} C_DIS
LIN {X -89.9473,Y 87.8239,Z 137,A 132.1974,B 24.9469,C -1.6836,E1 24.8845,E2 674.0352} C_DIS
LIN {X -92.9279,Y 84.6637,Z 137,A 134.1986,B 24.9471,C -1.6796,E1 24.8807,E2 672.0349} C_DIS
LIN {X -95.9645,Y 81.2057,Z 137,A 136.2514,B 24.9476,C -1.6721,E1 24.877,E2 669.9906} C_DIS
LIN {X -98.53,Y 78.0729,Z 137,A 138.1315,B 24.9478,C -1.6687,E1 24.8737,E2 668.1098} C_DIS
LIN {X -101.1145,Y 74.6956,Z 137,A 140.1303,B 24.948,C -1.6661,E1 24.8704,E2 666.1075} C_DIS
LIN {X -103.7946,Y 70.924,Z 137,A 142.2106,B 24.9484,C -1.6589,E1 24.867,E2 664.0342} C_DIS
LIN {X -106.1058,Y 67.4179,Z 137,A 144.1631,B 24.9487,C -1.6552,E1 24.8641,E2 662.0807} C_DIS
LIN {X -108.573,Y 63.3681,Z 137,A 146.5309,B 24.9485,C -1.6583,E1 24.8607,E2 659.6933} C_DIS
LIN {X -111.9906,Y 57.1062,Z 137,A 149.2935,B 24.9504,C -1.6264,E1 24.8571,E2 656.992} C_DIS
LIN {X -113.2459,Y 54.5762,Z 137,A 150.9211,B 24.9497,C -1.6379,E1 24.8551,E2 655.3283} C_DIS
LIN {X -114.9316,Y 50.9306,Z 137,A 152.737,B 24.9501,C -1.6316,E1 24.853,E2 653.5174} C_DIS
LIN {X -116.7204,Y 46.6849,Z 137,A 154.755,B 24.9507,C -1.6213,E1 24.8509,E2 651.5126} C_DIS
LIN {X -118.0073,Y 43.3344,Z 137,A 156.5195,B 24.9507,C -1.622,E1 24.8491,E2 649.7366} C_DIS
LIN {X -119.2357,Y 39.8235,Z 137,A 158.1333,B 24.9513,C -1.613,E1 24.8477,E2 648.1351} C_DIS
LIN {X -120.3671,Y 36.2645,Z 137,A 159.7915,B 24.9517,C -1.6055,E1 24.8463,E2 646.4851} C_DIS
LIN {X -121.4111,Y 32.5952,Z 137,A 161.5884,B 24.9519,C -1.6026,E1 24.845,E2 644.6848} C_DIS
LIN {X -122.6559,Y 27.5464,Z 137,A 164.0798,B 24.952,C -1.6004,E1 24.8434,E2 642.1841} C_DIS
LIN {X -123.5057,Y 23.4401,Z 137,A 165.8777,B 24.9527,C -1.589,E1 24.8424,E2 640.4026} C_DIS
LIN {X -124.1541,Y 19.7254,Z 137,A 167.9329,B 24.9521,C -1.5986,E1 24.8415,E2 638.3123} C_DIS
LIN {X -124.6167,Y 16.5477,Z 137,A 168.8216,B 24.9539,C -1.5679,E1 24.8412,E2 637.4916} C_DIS
LIN {X -124.9314,Y 13.9839,Z 137,A 170.5119,B 24.9528,C -1.5871,E1 24.8406,E2 635.7453} C_DIS
LIN {X -125.3654,Y 9.3097,Z 137,A 172.4995,B 24.9536,C -1.5732,E1 24.8401,E2 633.7788} C_DIS
LIN {X -125.6113,Y 4.9946,Z 137,A 174.491,B 24.954,C -1.5677,E1 24.8399,E2 631.7885} C_DIS
LIN {X -125.7119,Y 0.4141,Z 137,A 176.5121,B 24.9545,C -1.5578,E1 24.8398,E2 629.7789} C_DIS
LIN {X -125.6786,Y -2.8976,Z 137,A 178.1517,B 24.9545,C -1.5588,E1 24.8398,E2 628.1271} C_DIS
LIN {X -125.5287,Y -6.7744,Z 137,A 179.9603,B 24.9547,C -1.5548,E1 24.8401,E2 626.3171} C_DIS
LIN {X -125.1753,Y -11.5947,Z 137,A -177.9462,B 24.9554,C -1.5427,E1 24.8406,E2 624.2399} C_DIS
LIN {X -124.813,Y -14.9948,Z 137,A -176.4075,B 24.9558,C -1.5368,E1 24.8411,E2 622.7061} C_DIS
LIN {X -124.3141,Y -18.692,Z 137,A -174.3355,B 24.9551,C -1.5482,E1 24.8419,E2 620.5945} C_DIS
LIN {X -123.7738,Y -21.9808,Z 137,A -173.4304,B 24.957,C -1.5155,E1 24.8423,E2 619.762} C_DIS
LIN {X -123.155,Y -25.2181,Z 137,A -171.7221,B 24.9567,C -1.52,E1 24.8432,E2 618.0328} C_DIS
LIN {X -122.2649,Y -29.23,Z 137,A -170.0172,B 24.9575,C -1.5065,E1 24.8443,E2 616.3502} C_DIS
LIN {X -121.5832,Y -31.9497,Z 137,A -168.4018,B 24.9568,C -1.5178,E1 24.8454,E2 614.6983} C_DIS
LIN {X -120.627,Y -35.386,Z 137,A -166.8382,B 24.9573,C -1.5099,E1 24.8466,E2 613.1444} C_DIS
LIN {X -119.7096,Y -38.3755,Z 137,A -165.4037,B 24.9575,C -1.506,E1 24.8478,E2 611.711} C_DIS
LIN {X -118.4308,Y -42.1595,Z 137,A -163.42,B 24.9575,C -1.5079,E1 24.8497,E2 609.7115} C_DIS
LIN {X -117.0907,Y -45.7477,Z 137,A -161.7645,B 24.9579,C -1.4986,E1 24.8513,E2 608.0689} C_DIS
LIN {X -115.4933,Y -49.6425,Z 137,A -159.8166,B 24.9582,C -1.4943,E1 24.8534,E2 606.1204} C_DIS
LIN {X -114.0545,Y -52.864,Z 137,A -158.1356,B 24.9582,C -1.493,E1 24.8554,E2 604.4334} C_DIS
LIN {X -112.4889,Y -56.1211,Z 137,A -156.4788,B 24.9585,C -1.4887,E1 24.8574,E2 602.7778} C_DIS
LIN {X -110.53,Y -59.8893,Z 137,A -154.5332,B 24.9588,C -1.4837,E1 24.86,E2 600.8337} C_DIS
LIN {X -108.2987,Y -63.8349,Z 137,A -152.519,B 24.9592,C -1.4757,E1 24.8628,E2 598.8281} C_DIS
LIN {X -105.6191,Y -68.1777,Z 137,A -150.2783,B 24.9598,C -1.4656,E1 24.8661,E2 596.6002} C_DIS
LIN {X -103.4519,Y -71.4234,Z 137,A -148.637,B 24.9604,C -1.4546,E1 24.8686,E2 594.9768} C_DIS
LIN {X -101.7448,Y -73.8341,Z 137,A -146.9767,B 24.9598,C -1.4657,E1 24.8714,E2 593.282} C_DIS
LIN {X -99.3499,Y -77.0265,Z 137,A -145.1858,B 24.9601,C -1.4599,E1 24.8744,E2 591.4963} C_DIS
LIN {X -96.5939,Y -80.4563,Z 137,A -143.1695,B 24.9603,C -1.4556,E1 24.878,E2 589.4809} C_DIS
LIN {X -93.7025,Y -83.8052,Z 137,A -141.308,B 24.961,C -1.4437,E1 24.8813,E2 587.6393} C_DIS
LIN {X -91.2153,Y -86.5064,Z 137,A -139.4668,B 24.9607,C -1.4478,E1 24.8849,E2 585.7805} C_DIS
LIN {X -88.2914,Y -89.4888,Z 137,A -137.5257,B 24.9609,C -1.4454,E1 24.8887,E2 583.8367} C_DIS
LIN {X -85.41,Y -92.2428,Z 137,A -135.742,B 24.9612,C -1.4401,E1 24.8923,E2 582.0584} C_DIS
LIN {X -82.3295,Y -95.0025,Z 137,A -133.7972,B 24.9612,C -1.4391,E1 24.8964,E2 580.1082} C_DIS
LIN {X -78.6033,Y -98.1079,Z 137,A -131.5643,B 24.9614,C -1.436,E1 24.9013,E2 577.8744} C_DIS
LIN {X -75.1089,Y -100.8074,Z 137,A -129.7525,B 24.9621,C -1.4229,E1 24.9052,E2 576.0872} C_DIS
LIN {X -72.1791,Y -102.926,Z 137,A -127.9041,B 24.9617,C -1.4295,E1 24.9095,E2 574.2166} C_DIS
LIN {X -68.5713,Y -105.3635,Z 137,A -125.169,B 24.9599,C -1.4622,E1 24.9161,E2 571.3949} C_DIS
LIN {X -63.5374,Y -108.4734,Z 137,A -123.4216,B 24.9626,C -1.4127,E1 24.92,E2 569.7597} C_DIS
LIN {X -61.1582,Y -109.8328,Z 137,A -121.9787,B 24.9622,C -1.4202,E1 24.9236,E2 568.2949} C_DIS
LIN {X -58.2505,Y -111.3999,Z 137,A -120.5615,B 24.9625,C -1.414,E1 24.927,E2 566.8885} C_DIS
LIN {X -55.0912,Y -112.9969,Z 137,A -118.8306,B 24.9624,C -1.4176,E1 24.9314,E2 565.1446} C_DIS
LIN {X -51.3861,Y -114.7279,Z 137,A -117.0902,B 24.9628,C -1.4095,E1 24.9358,E2 563.4189} C_DIS
LIN {X -48.3861,Y -116.025,Z 137,A -115.5708,B 24.9628,C -1.4093,E1 24.9397,E2 561.8965} C_DIS
LIN {X -44.8666,Y -117.4332,Z 137,A -113.722,B 24.9626,C -1.4134,E1 24.9446,E2 560.034} C_DIS
LIN {X -40.7212,Y -118.933,Z 137,A -111.9402,B 24.9632,C -1.4007,E1 24.9492,E2 558.2788} C_DIS
LIN {X -38.2287,Y -119.7565,Z 137,A -110.6774,B 24.9632,C -1.403,E1 24.9525,E2 557.0083} C_DIS
LIN {X -35.1856,Y -120.6857,Z 137,A -109.1883,B 24.9631,C -1.4038,E1 24.9565,E2 555.5148} C_DIS
LIN {X -31.8366,Y -121.6134,Z 137,A -107.4166,B 24.9627,C -1.412,E1 24.9614,E2 553.7211} C_DIS
LIN {X -28.137,Y -122.521,Z 137,A -105.8657,B 24.9632,C -1.402,E1 24.9655,E2 552.1917} C_DIS
LIN {X -25.0145,Y -123.1964,Z 137,A -104.434,B 24.9632,C -1.4002,E1 24.9694,E2 550.7626} C_DIS
LIN {X -21.5393,Y -123.8528,Z 137,A -102.6762,B 24.9629,C -1.4067,E1 24.9743,E2 548.9876} C_DIS
LIN {X -17.7279,Y -124.4541,Z 137,A -101.0457,B 24.9633,C -1.4,E1 24.9788,E2 547.3716} C_DIS
LIN {X -13.8071,Y -124.9504,Z 137,A -99.1963,B 24.9632,C -1.4021,E1 24.9839,E2 545.516} C_DIS
LIN {X -9.9677,Y -125.3162,Z 137,A -97.3474,B 24.9629,C -1.4065,E1 24.9891,E2 543.6559} C_DIS
LIN {X -6.0444,Y -125.5654,Z 137,A -95.6022,B 24.9631,C -1.4043,E1 24.994,E2 541.9154} C_DIS
LIN {X -2.0834,Y -125.6933,Z 137,A -93.8318,B 24.9631,C -1.4028,E1 24.9989,E2 540.1484} C_DIS
LIN {X 0.8908,Y -125.7045,Z 137,A -92.7626,B 24.9639,C -1.389,E1 25.0018,E2 539.1117} C_DIS
Enddeposition()
LIN {X 0.8908,Y -125.7045,Z 137,A -92.7626,B 24.9639,C -1.389,E1 25.0018,E2 539.1117} C_DIS
Startdeposition()
$VEL.CP = VEL_PRINT
LIN {X -0.7216,Y -124.7233,Z 137,A -94.0282,B 24.9643,C -1.3805,E1 24.9982,E2 540.3975} C_DIS
LIN {X -4.8668,Y -124.6303,Z 137,A -95.9194,B 24.9643,C -1.3809,E1 24.9929,E2 542.288} C_DIS
LIN {X -8.9163,Y -124.4063,Z 137,A -97.7628,B 24.9643,C -1.3818,E1 24.9878,E2 544.1299} C_DIS
LIN {X -12.7212,Y -124.0764,Z 137,A -99.5785,B 24.9643,C -1.379,E1 24.9827,E2 545.9533} C_DIS
LIN {X -16.3827,Y -123.6447,Z 137,A -101.2456,B 24.9643,C -1.3806,E1 24.9781,E2 547.6178} C_DIS
LIN {X -20.3553,Y -123.053,Z 137,A -103.0805,B 24.9643,C -1.3816,E1 24.973,E2 549.4519} C_DIS
LIN {X -24.2187,Y -122.353,Z 137,A -105.0981,B 24.9647,C -1.3721,E1 24.9674,E2 551.4942} C_DIS
LIN {X -28.5228,Y -121.422,Z 137,A -107.354,B 24.9652,C -1.3621,E1 24.9612,E2 553.7768} C_DIS
LIN {X -32.2345,Y -120.4877,Z 137,A -108.6476,B 24.9641,C -1.3851,E1 24.9579,E2 555.0177} C_DIS
LIN {X -36.1679,Y -119.3663,Z 137,A -110.6925,B 24.9644,C -1.3786,E1 24.9524,E2 557.0814} C_DIS
LIN {X -40.8612,Y -117.8417,Z 137,A -112.8613,B 24.9641,C -1.3851,E1 24.9466,E2 559.2388} C_DIS
LIN {X -44.6396,Y -116.4644,Z 137,A -114.7445,B 24.9641,C -1.3851,E1 24.9417,E2 561.1258} C_DIS
LIN {X -48.1702,Y -115.0475,Z 137,A -116.3975,B 24.9637,C -1.3914,E1 24.9375,E2 562.7677} C_DIS
LIN {X -51.6762,Y -113.5183,Z 137,A -118.2897,B 24.964,C -1.387,E1 24.9326,E2 564.6748} C_DIS
LIN {X -55.1164,Y -111.8859,Z 137,A -119.8999,B 24.9635,C -1.3957,E1 24.9286,E2 566.2686} C_DIS
LIN {X -57.6064,Y -110.6253,Z 137,A -121.2548,B 24.9636,C -1.3939,E1 24.9252,E2 567.6313} C_DIS
LIN {X -61.3318,Y -108.6058,Z 137,A -123.2336,B 24.9636,C -1.3951,E1 24.9204,E2 569.6131} C_DIS
LIN {X -65.9299,Y -105.8772,Z 137,A -125.7004,B 24.9634,C -1.3983,E1 24.9145,E2 572.0798} C_DIS
LIN {X -69.5955,Y -103.5054,Z 137,A -127.5092,B 24.9627,C -1.4106,E1 24.9103,E2 573.8653} C_DIS
LIN {X -72.5763,Y -101.4368,Z 137,A -129.1397,B 24.9625,C -1.4151,E1 24.9066,E2 575.4907} C_DIS
LIN {X -75.2427,Y -99.4751,Z 137,A -130.9151,B 24.963,C -1.4061,E1 24.9025,E2 577.2938} C_DIS
LIN {X -78.1193,Y -97.2326,Z 137,A -132.9822,B 24.9637,C -1.3913,E1 24.8979,E2 579.4037} C_DIS
LIN {X -81.1715,Y -94.6996,Z 137,A -134.4558,B 24.9627,C -1.4108,E1 24.8949,E2 580.8368} C_DIS
LIN {X -84.5086,Y -91.7336,Z 137,A -136.1915,B 24.9617,C -1.4293,E1 24.8914,E2 582.5352} C_DIS
LIN {X -87.3422,Y -89.0398,Z 137,A -138.2652,B 24.9622,C -1.4204,E1 24.8871,E2 584.6388} C_DIS
LIN {X -90.3654,Y -85.9705,Z 137,A -140.2656,B 24.962,C -1.4238,E1 24.8832,E2 586.6398} C_DIS
LIN {X -92.4516,Y -83.7225,Z 137,A -142.1242,B 24.9629,C -1.4067,E1 24.8797,E2 588.5473} C_DIS
LIN {X -95.2073,Y -80.5754,Z 137,A -143.6329,B 24.9617,C -1.4298,E1 24.877,E2 590.0079} C_DIS
LIN {X -97.8562,Y -77.3373,Z 137,A -145.8701,B 24.9622,C -1.4203,E1 24.8731,E2 592.2783} C_DIS
LIN {X -100.0259,Y -74.5088,Z 137,A -147.1493,B 24.9611,C -1.4405,E1 24.871,E2 593.5156} C_DIS
LIN {X -102.3473,Y -71.2865,Z 137,A -148.9848,B 24.9609,C -1.4446,E1 24.868,E2 595.3502} C_DIS
LIN {X -104.2955,Y -68.4049,Z 137,A -150.4928,B 24.9605,C -1.4528,E1 24.8657,E2 596.8462} C_DIS
LIN {X -106.5247,Y -64.8798,Z 137,A -152.6251,B 24.9607,C -1.4482,E1 24.8625,E2 599.0003} C_DIS
LIN {X -108.818,Y -60.9543,Z 137,A -154.6784,B 24.9603,C -1.4555,E1 24.8597,E2 601.0469} C_DIS
LIN {X -110.7412,Y -57.3858,Z 137,A -156.5883,B 24.9601,C -1.4586,E1 24.8572,E2 602.9597} C_DIS
LIN {X -112.2539,Y -54.3672,Z 137,A -158.6014,B 24.961,C -1.4425,E1 24.8547,E2 605.022} C_DIS
LIN {X -114.1365,Y -50.2954,Z 137,A -160.2224,B 24.9596,C -1.4679,E1 24.8529,E2 606.5913} C_DIS
LIN {X -115.5922,Y -46.8486,Z 137,A -161.8548,B 24.9591,C -1.4769,E1 24.8512,E2 608.2114} C_DIS
LIN {X -117.3809,Y -42.1669,Z 137,A -164.1583,B 24.9588,C -1.4837,E1 24.8489,E2 610.5116} C_DIS
LIN {X -118.6586,Y -38.4279,Z 137,A -166.0125,B 24.9585,C -1.4875,E1 24.8473,E2 612.3674} C_DIS
LIN {X -119.6937,Y -35.0678,Z 137,A -167.5966,B 24.9582,C -1.4939,E1 24.846,E2 613.9456} C_DIS
LIN {X -120.7178,Y -31.3696,Z 137,A -169.4901,B 24.9582,C -1.4935,E1 24.8446,E2 615.8508} C_DIS
LIN {X -121.4796,Y -28.2719,Z 137,A -171.282,B 24.9588,C -1.4837,E1 24.8435,E2 617.6766} C_DIS
LIN {X -122.2732,Y -24.6106,Z 137,A -172.6085,B 24.9575,C -1.5066,E1 24.8427,E2 618.9565} C_DIS
LIN {X -123.4408,Y -17.8546,Z 137,A -175.7643,B 24.9569,C -1.5164,E1 24.8413,E2 622.1077} C_DIS
LIN {X -123.9363,Y -14.0229,Z 137,A -177.4689,B 24.9564,C -1.5252,E1 24.8407,E2 623.8015} C_DIS
LIN {X -124.3497,Y -9.6906,Z 137,A -179.9602,B 24.9573,C -1.51,E1 24.8401,E2 626.3438} C_DIS
LIN {X -124.5745,Y -6.1324,Z 137,A 178.72,B 24.9562,C -1.5293,E1 24.8399,E2 627.6255} C_DIS
LIN {X -124.7026,Y -2.4042,Z 137,A 176.7651,B 24.9565,C -1.5243,E1 24.8398,E2 629.6041} C_DIS
LIN {X -124.7237,Y 0.8284,Z 137,A 175.0397,B 24.9568,C -1.5187,E1 24.8398,E2 631.3533} C_DIS
LIN {X -124.6231,Y 5.053,Z 137,A 173.592,B 24.9552,C -1.5467,E1 24.84,E2 632.7431} C_DIS
LIN {X -124.3737,Y 9.3629,Z 137,A 170.9876,B 24.9564,C -1.526,E1 24.8405,E2 635.4123} C_DIS
LIN {X -123.9199,Y 14.1639,Z 137,A 169.4926,B 24.9541,C -1.5648,E1 24.8409,E2 636.8239} C_DIS
LIN {X -122.9545,Y 20.9459,Z 137,A 166.2522,B 24.9538,C -1.5709,E1 24.8423,E2 640.069} C_DIS
LIN {X -121.2005,Y 29.4419,Z 137,A 162.2104,B 24.9531,C -1.5814,E1 24.8446,E2 644.1098} C_DIS
LIN {X -120.1944,Y 33.3123,Z 137,A 160.3523,B 24.9528,C -1.5863,E1 24.8459,E2 645.9668} C_DIS
LIN {X -118.9003,Y 37.6713,Z 137,A 158.326,B 24.9523,C -1.5958,E1 24.8476,E2 647.9822} C_DIS
LIN {X -118.0164,Y 40.3575,Z 137,A 156.8902,B 24.9524,C -1.5939,E1 24.8488,E2 649.4309} C_DIS
LIN {X -116.879,Y 43.539,Z 137,A 155.3631,B 24.952,C -1.5999,E1 24.8503,E2 650.9523} C_DIS
LIN {X -114.7295,Y 48.9266,Z 137,A 152.6444,B 24.9517,C -1.6057,E1 24.8532,E2 653.6721} C_DIS
LIN {X -113.5339,Y 51.6402,Z 137,A 151.0765,B 24.952,C -1.6009,E1 24.855,E2 655.2602} C_DIS
LIN {X -111.4113,Y 56.0725,Z 137,A 148.642,B 24.952,C -1.5999,E1 24.858,E2 657.71} C_DIS
LIN {X -109.683,Y 59.3827,Z 137,A 147.4248,B 24.9504,C -1.627,E1 24.8596,E2 658.8692} C_DIS
LIN {X -108.5199,Y 61.4842,Z 137,A 145.6281,B 24.9521,C -1.5997,E1 24.8622,E2 660.7403} C_DIS
LIN {X -106.204,Y 65.4025,Z 137,A 144.0325,B 24.9504,C -1.6276,E1 24.8644,E2 662.2778} C_DIS
LIN {X -103.9856,Y 68.8756,Z 137,A 142.1576,B 24.95,C -1.6338,E1 24.8672,E2 664.1473} C_DIS
LIN {X -101.3644,Y 72.6776,Z 137,A 140.0607,B 24.9496,C -1.6408,E1 24.8706,E2 666.2378} C_DIS
LIN {X -98.851,Y 76.0615,Z 137,A 138.012,B 24.9496,C -1.6411,E1 24.874,E2 668.2956} C_DIS
LIN {X -96.1269,Y 79.4756,Z 137,A 136.0287,B 24.9491,C -1.6475,E1 24.8775,E2 670.2728} C_DIS
LIN {X -93.3118,Y 82.7629,Z 137,A 134.0154,B 24.9489,C -1.6516,E1 24.8812,E2 672.2856} C_DIS
LIN {X -90.4278,Y 85.9052,Z 137,A 132.0142,B 24.9487,C -1.6546,E1 24.885,E2 674.2883} C_DIS
LIN {X -87.2989,Y 89.0822,Z 137,A 130.0061,B 24.9483,C -1.6615,E1 24.889,E2 676.2885} C_DIS
LIN {X -84.1198,Y 92.091,Z 137,A 127.9342,B 24.9481,C -1.6635,E1 24.8932,E2 678.3641} C_DIS
LIN {X -80.8427,Y 94.98,Z 137,A 125.9716,B 24.9477,C -1.6701,E1 24.8973,E2 680.3186} C_DIS
LIN {X -77.3786,Y 97.8235,Z 137,A 123.855,B 24.9477,C -1.6721,E1 24.9019,E2 682.4385} C_DIS
LIN {X -73.9807,Y 100.4172,Z 137,A 121.9612,B 24.9471,C -1.6794,E1 24.9062,E2 684.3217} C_DIS
LIN {X -70.6876,Y 102.762,Z 137,A 120.053,B 24.9471,C -1.6809,E1 24.9105,E2 686.2328} C_DIS
LIN {X -66.9834,Y 105.2144,Z 137,A 118.004,B 24.9468,C -1.6845,E1 24.9153,E2 688.2799} C_DIS
LIN {X -63.869,Y 107.1331,Z 137,A 115.3911,B 24.9492,C -1.6458,E1 24.9219,E2 690.9928} C_DIS
LIN {X -58.1771,Y 110.3256,Z 137,A 113.6596,B 24.9453,C -1.7081,E1 24.9257,E2 692.5811} C_DIS
LIN {X -53.8633,Y 112.4946,Z 137,A 110.6635,B 24.9473,C -1.6763,E1 24.9335,E2 695.6606} C_DIS
LIN {X -50.0227,Y 114.2556,Z 137,A 109.3394,B 24.9454,C -1.7073,E1 24.9367,E2 696.9143} C_DIS
LIN {X -47.1669,Y 115.4639,Z 137,A 107.7845,B 24.9456,C -1.7033,E1 24.9407,E2 698.4821} C_DIS
LIN {X -44.111,Y 116.6648,Z 137,A 106.2426,B 24.9456,C -1.7039,E1 24.9447,E2 700.026} C_DIS
LIN {X -41.1804,Y 117.7311,Z 137,A 104.649,B 24.9459,C -1.6983,E1 24.9489,E2 701.6359} C_DIS
LIN {X -35.65,Y 119.5232,Z 137,A 102.0835,B 24.9454,C -1.7062,E1 24.9557,E2 704.1871} C_DIS
LIN {X -31.9191,Y 120.5718,Z 137,A 99.7169,B 24.947,C -1.6812,E1 24.9623,E2 706.6167} C_DIS
LIN {X -27.106,Y 121.7449,Z 137,A 97.6358,B 24.9463,C -1.6922,E1 24.9679,E2 708.6744} C_DIS
LIN {X -23.2711,Y 122.535,Z 137,A 96.3078,B 24.9449,C -1.7154,E1 24.9714,E2 709.9487} C_DIS
LIN {X -19.3783,Y 123.2109,Z 137,A 94.5882,B 24.9445,C -1.7212,E1 24.9761,E2 711.6563} C_DIS
LIN {X -16.0661,Y 123.6862,Z 137,A 92.8898,B 24.9449,C -1.7147,E1 24.9808,E2 713.3716} C_DIS
LIN {X -11.8661,Y 124.1595,Z 137,A 90.9801,B 24.9447,C -1.7172,E1 24.9861,E2 715.2763} C_DIS
LIN {X -7.8726,Y 124.4768,Z 137,A 89.1439,B 24.9447,C -1.7182,E1 24.9912,E2 717.1109} C_DIS
LIN {X -4.0185,Y 124.6618,Z 137,A 87.3368,B 24.9447,C -1.7171,E1 24.9963,E2 718.9209} C_DIS
LIN {X -0.47,Y 124.7247,Z 137,A 85.7737,B 24.9445,C -1.7207,E1 25.0006,E2 720.4756} C_DIS
LIN {X 3.4119,Y 124.6787,Z 137,A 83.9517,B 24.9446,C -1.7191,E1 25.0057,E2 722.3011} C_DIS
LIN {X 7.4483,Y 124.5029,Z 137,A 82.0947,B 24.9446,C -1.7191,E1 25.0109,E2 724.1574} C_DIS
LIN {X 11.2669,Y 124.217,Z 137,A 80.2581,B 24.9449,C -1.7153,E1 25.016,E2 726.0021} C_DIS
LIN {X 14.957,Y 123.8253,Z 137,A 78.6013,B 24.9447,C -1.7173,E1 25.0206,E2 727.653} C_DIS
LIN {X 18.8809,Y 123.2879,Z 137,A 76.8223,B 24.9447,C -1.7187,E1 25.0255,E2 729.4271} C_DIS
LIN {X 23.6716,Y 122.4584,Z 137,A 74.5655,B 24.9447,C -1.7167,E1 25.0317,E2 731.686} C_DIS
LIN {X 29.4881,Y 121.1894,Z 137,A 71.8102,B 24.9449,C -1.7143,E1 25.0393,E2 734.4433} C_DIS
LIN {X 33.0174,Y 120.2769,Z 137,A 70.0026,B 24.9454,C -1.7068,E1 25.0442,E2 736.2658} C_DIS
LIN {X 37.249,Y 119.0352,Z 137,A 68.1278,B 24.945,C -1.7125,E1 25.0491,E2 738.1238} C_DIS
LIN {X 40.4146,Y 117.9965,Z 137,A 66.7311,B 24.9447,C -1.7177,E1 25.0528,E2 739.5057} C_DIS
LIN {X 43.5164,Y 116.8875,Z 137,A 65.1868,B 24.9449,C -1.7147,E1 25.0568,E2 741.0536} C_DIS
LIN {X 46.4303,Y 115.7608,Z 137,A 63.7135,B 24.9451,C -1.7114,E1 25.0607,E2 742.5314} C_DIS
LIN {X 49.4888,Y 114.4864,Z 137,A 62.1802,B 24.9453,C -1.7092,E1 25.0646,E2 744.0664} C_DIS
LIN {X 52.7425,Y 113.0252,Z 137,A 60.5613,B 24.9453,C -1.7082,E1 25.0687,E2 745.6836} C_DIS
LIN {X 56.513,Y 111.1871,Z 137,A 58.6614,B 24.9453,C -1.7071,E1 25.0735,E2 747.581} C_DIS
LIN {X 59.6173,Y 109.5561,Z 137,A 56.6962,B 24.9466,C -1.6876,E1 25.0784,E2 749.5868} C_DIS
LIN {X 62.4744,Y 107.9522,Z 137,A 55.2775,B 24.9466,C -1.6896,E1 25.0818,E2 750.9965} C_DIS
LIN {X 66.8631,Y 105.291,Z 137,A 53.2836,B 24.9456,C -1.7037,E1 25.0865,E2 752.9506} C_DIS
LIN {X 69.7831,Y 103.3784,Z 137,A 51.4776,B 24.9464,C -1.6911,E1 25.0907,E2 754.7804} C_DIS
LIN {X 73.1394,Y 101.0315,Z 137,A 49.6508,B 24.9464,C -1.6905,E1 25.0949,E2 756.6022} C_DIS
LIN {X 75.4569,Y 99.3134,Z 137,A 48.1507,B 24.9471,C -1.6795,E1 25.0983,E2 758.1229} C_DIS
LIN {X 79.2975,Y 96.2744,Z 137,A 46.0159,B 24.9471,C -1.6809,E1 25.1029,E2 760.2465} C_DIS
LIN {X 82.8571,Y 93.2285,Z 137,A 43.8824,B 24.9473,C -1.6775,E1 25.1074,E2 762.3796} C_DIS
LIN {X 86.034,Y 90.3046,Z 137,A 41.9555,B 24.9473,C -1.6761,E1 25.1113,E2 764.3017} C_DIS
LIN {X 89.0022,Y 87.3806,Z 137,A 40.041,B 24.9476,C -1.672,E1 25.1151,E2 766.218} C_DIS
LIN {X 92.5945,Y 83.565,Z 137,A 37.6165,B 24.948,C -1.6656,E1 25.1197,E2 768.6468} C_DIS
LIN {X 95.4153,Y 80.3287,Z 137,A 35.6926,B 24.9482,C -1.6634,E1 25.1232,E2 770.5673} C_DIS
LIN {X 97.936,Y 77.2356,Z 137,A 33.8456,B 24.9485,C -1.6582,E1 25.1264,E2 772.4178} C_DIS
LIN {X 100.0621,Y 74.4602,Z 137,A 32.1018,B 24.9492,C -1.6473,E1 25.1294,E2 774.1791} C_DIS
LIN {X 103.0546,Y 70.2612,Z 137,A 29.7877,B 24.9494,C -1.6439,E1 25.133,E2 776.4898} C_DIS
LIN {X 105.6903,Y 66.2303,Z 137,A 27.6506,B 24.9494,C -1.6418,E1 25.1363,E2 778.6211} C_DIS
LIN {X 107.9927,Y 62.4046,Z 137,A 25.6437,B 24.9497,C -1.6385,E1 25.1391,E2 780.6256} C_DIS
LIN {X 110.0828,Y 58.6394,Z 137,A 23.7841,B 24.9497,C -1.639,E1 25.1416,E2 782.4743} C_DIS
LIN {X 112.2931,Y 54.2851,Z 137,A 21.2552,B 24.9509,C -1.6181,E1 25.1448,E2 785.0388} C_DIS
LIN {X 114.3958,Y 49.6984,Z 137,A 19.2104,B 24.9505,C -1.6252,E1 25.1471,E2 787.0557} C_DIS
LIN {X 115.7353,Y 46.4937,Z 137,A 17.6977,B 24.9505,C -1.6247,E1 25.1487,E2 788.5613} C_DIS
LIN {X 117.0715,Y 43.025,Z 137,A 15.8329,B 24.9513,C -1.6116,E1 25.1505,E2 790.4467} C_DIS
LIN {X 118.6432,Y 38.476,Z 137,A 13.1978,B 24.953,C -1.5834,E1 25.1529,E2 793.1334} C_DIS
LIN {X 119.9463,Y 34.1996,Z 137,A 11.6258,B 24.9519,C -1.6014,E1 25.1541,E2 794.6539} C_DIS
LIN {X 121.0785,Y 29.948,Z 137,A 9.0824,B 24.9539,C -1.5686,E1 25.1558,E2 797.26} C_DIS
LIN {X 122.1223,Y 25.3523,Z 137,A 7.5657,B 24.9524,C -1.5946,E1 25.1567,E2 798.7065} C_DIS
LIN {X 122.7464,Y 22.1294,Z 137,A 6.0584,B 24.9526,C -1.5899,E1 25.1574,E2 800.2162} C_DIS
LIN {X 123.3498,Y 18.4813,Z 137,A 4.2576,B 24.9533,C -1.5792,E1 25.1582,E2 802.0316} C_DIS
LIN {X 123.8655,Y 14.6194,Z 137,A 2.6146,B 24.9532,C -1.5809,E1 25.1588,E2 803.6608} C_DIS
LIN {X 124.2321,Y 11.0963,Z 137,A 0.9006,B 24.9537,C -1.5712,E1 25.1593,E2 805.3876} C_DIS
LIN {X 124.5059,Y 7.3991,Z 137,A -0.8032,B 24.9541,C -1.5656,E1 25.1596,E2 807.0945} C_DIS
LIN {X 124.6788,Y 3.4083,Z 137,A -2.5148,B 24.9541,C -1.5659,E1 25.1598,E2 808.7952} C_DIS
LIN {X 124.7289,Y 0,Z 137,A -4.2711,B 24.9549,C -1.5509,E1 25.1598,E2 810.5763} C_DIS
LIN {X 124.6526,Y -4.2957,Z 137,A -6.131,B 24.9549,C -1.5503,E1 25.1596,E2 812.4266} C_DIS
LIN {X 124.4692,Y -7.996,Z 137,A -7.7698,B 24.9551,C -1.5479,E1 25.1594,E2 814.0612} C_DIS
LIN {X 124.1706,Y -11.7504,Z 137,A -9.4189,B 24.9551,C -1.5464,E1 25.159,E2 815.7042} C_DIS
LIN {X 123.7555,Y -15.5375,Z 137,A -11.2767,B 24.9559,C -1.5351,E1 25.1584,E2 817.5776} C_DIS
LIN {X 123.2406,Y -19.1866,Z 137,A -12.8873,B 24.9559,C -1.5338,E1 25.1577,E2 819.1818} C_DIS
LIN {X 122.5843,Y -23.0134,Z 137,A -14.6905,B 24.9563,C -1.5269,E1 25.1568,E2 820.9906} C_DIS
LIN {X 122.0293,Y -25.797,Z 137,A -16.9295,B 24.9592,C -1.475,E1 25.1555,E2 823.3389} C_DIS
LIN {X 120.5217,Y -32.1069,Z 137,A -18.5905,B 24.956,C -1.5327,E1 25.1544,E2 824.8544} C_DIS
LIN {X 118.6889,Y -38.333,Z 137,A -21.8079,B 24.9572,C -1.5109,E1 25.1518,E2 828.1049} C_DIS
LIN {X 117.647,Y -41.4228,Z 137,A -23.3707,B 24.9577,C -1.5028,E1 25.1504,E2 829.678} C_DIS
LIN {X 116.3358,Y -44.9703,Z 137,A -25.1031,B 24.958,C -1.4976,E1 25.1487,E2 831.4131} C_DIS
LIN {X 113.9443,Y -50.725,Z 137,A -27.9089,B 24.9583,C -1.4916,E1 25.1456,E2 834.2176} C_DIS
LIN {X 112.5098,Y -53.8315,Z 137,A -29.4339,B 24.9585,C -1.4891,E1 25.1438,E2 835.74} C_DIS
LIN {X 111.2084,Y -56.4712,Z 137,A -30.8053,B 24.9587,C -1.484,E1 25.1421,E2 837.1162} C_DIS
LIN {X 109.5967,Y -59.5428,Z 137,A -32.2449,B 24.9586,C -1.4871,E1 25.1402,E2 838.541} C_DIS
LIN {X 107.8229,Y -62.6979,Z 137,A -34.1039,B 24.9594,C -1.4721,E1 25.1376,E2 840.4257} C_DIS
LIN {X 105.7298,Y -66.1669,Z 137,A -35.9921,B 24.9598,C -1.4653,E1 25.1349,E2 842.3204} C_DIS
LIN {X 103.4417,Y -69.6895,Z 137,A -37.9157,B 24.9601,C -1.46,E1 25.1319,E2 844.2467} C_DIS
LIN {X 101.0066,Y -73.1738,Z 137,A -39.8525,B 24.9603,C -1.4554,E1 25.1288,E2 846.185} C_DIS
LIN {X 98.8343,Y -76.0833,Z 137,A -41.3757,B 24.9602,C -1.4581,E1 25.1262,E2 847.6946} C_DIS
LIN {X 96.4513,Y -79.0817,Z 137,A -43.6724,B 24.9619,C -1.4262,E1 25.1221,E2 850.056} C_DIS
LIN {X 93.7751,Y -82.2379,Z 137,A -45.1445,B 24.961,C -1.4428,E1 25.1194,E2 851.4821} C_DIS
LIN {X 88.8392,Y -87.5467,Z 137,A -48.3196,B 24.961,C -1.4422,E1 25.1134,E2 854.6449} C_DIS
LIN {X 85.1509,Y -91.1378,Z 137,A -50.8294,B 24.9617,C -1.4291,E1 25.1083,E2 857.1753} C_DIS
LIN {X 83.1248,Y -92.9894,Z 137,A -52.3959,B 24.9627,C -1.4107,E1 25.105,E2 858.7788} C_DIS
LIN {X 80.341,Y -95.4045,Z 137,A -53.8612,B 24.9623,C -1.4182,E1 25.1019,E2 860.2207} C_DIS
LIN {X 76.6241,Y -98.4153,Z 137,A -55.9345,B 24.9623,C -1.4196,E1 25.0974,E2 862.283} C_DIS
LIN {X 73.2597,Y -100.9444,Z 137,A -57.8669,B 24.9625,C -1.4155,E1 25.093,E2 864.2182} C_DIS
LIN {X 68.4737,Y -104.2502,Z 137,A -60.4759,B 24.9625,C -1.4132,E1 25.087,E2 866.8237} C_DIS
LIN {X 64.8958,Y -106.5149,Z 137,A -62.4996,B 24.963,C -1.4055,E1 25.0822,E2 868.8592} C_DIS
LIN {X 59.152,Y -109.8081,Z 137,A -65.5642,B 24.9633,C -1.3989,E1 25.0747,E2 871.9305} C_DIS
LIN {X 55.316,Y -111.7875,Z 137,A -67.3771,B 24.9631,C -1.404,E1 25.0702,E2 873.7263} C_DIS
LIN {X 52.4817,Y -113.1458,Z 137,A -68.8157,B 24.9631,C -1.4019,E1 25.0666,E2 875.1661} C_DIS
LIN {X 49.8259,Y -114.3407,Z 137,A -70.2819,B 24.9636,C -1.3935,E1 25.0628,E2 876.6486} C_DIS
LIN {X 45.8934,Y -115.977,Z 137,A -72.2544,B 24.9638,C -1.3898,E1 25.0577,E2 878.6252} C_DIS
LIN {X 41.0866,Y -117.7636,Z 137,A -74.5844,B 24.9639,C -1.388,E1 25.0516,E2 880.9548} C_DIS
LIN {X 36.0679,Y -119.3969,Z 137,A -77.4049,B 24.9651,C -1.3657,E1 25.0439,E2 883.8231} C_DIS
LIN {X 31.9992,Y -120.5504,Z 137,A -78.8385,B 24.9639,C -1.3885,E1 25.0402,E2 885.2004} C_DIS
LIN {X 28.2732,Y -121.4793,Z 137,A -80.9,B 24.9647,C -1.3722,E1 25.0345,E2 887.2976} C_DIS
LIN {X 25.1248,Y -122.1686,Z 137,A -82.1872,B 24.9643,C -1.3803,E1 25.0311,E2 888.5639} C_DIS
LIN {X 20.5868,Y -123.0144,Z 137,A -84.1817,B 24.9641,C -1.3847,E1 25.0256,E2 890.5457} C_DIS
LIN {X 16.582,Y -123.6186,Z 137,A -86.0646,B 24.9642,C -1.3823,E1 25.0204,E2 892.4325} C_DIS
LIN {X 13.4946,Y -123.9931,Z 137,A -87.5274,B 24.9643,C -1.3798,E1 25.0163,E2 893.9004} C_DIS
LIN {X 9.2334,Y -124.3831,Z 137,A -89.4527,B 24.9643,C -1.3808,E1 25.011,E2 895.8222} C_DIS
LIN {X 5.0872,Y -124.6217,Z 137,A -91.3425,B 24.9643,C -1.3809,E1 25.0057,E2 897.7112} C_DIS
LIN {X 0.8894,Y -124.721,Z 137,A -93.1958,B 24.9641,C -1.384,E1 25.0005,E2 899.5568} C_DIS
Enddeposition()
LIN {X 0.8894,Y -124.721,Z 137,A -93.1958,B 24.9641,C -1.384,E1 25.0005,E2 899.5568} C_DIS
Startdeposition()
$VEL.CP = VEL_PRINT
LIN {X 2.1859,Y -123.7209,Z 137,A -91.9732,B 24.9616,C -1.4316,E1 25.0043,E2 898.2217} C_DIS
LIN {X 6.2094,Y -123.5842,Z 137,A -90.1344,B 24.9616,C -1.431,E1 25.0094,E2 896.3847} C_DIS
LIN {X 10.0711,Y -123.33,Z 137,A -88.2898,B 24.9615,C -1.4344,E1 25.0146,E2 894.5329} C_DIS
LIN {X 13.9112,Y -122.9574,Z 137,A -86.4272,B 24.9612,C -1.4392,E1 25.0198,E2 892.6603} C_DIS
LIN {X 17.553,Y -122.4887,Z 137,A -84.8321,B 24.9614,C -1.4352,E1 25.0241,E2 891.076} C_DIS
LIN {X 21.1412,Y -121.9224,Z 137,A -83.0811,B 24.9612,C -1.4399,E1 25.029,E2 889.3158} C_DIS
LIN {X 27.4048,Y -120.6671,Z 137,A -79.75,B 24.96,C -1.461,E1 25.0382,E2 885.9388} C_DIS
LIN {X 31.3134,Y -119.7137,Z 137,A -78.4641,B 24.9615,C -1.4343,E1 25.0415,E2 884.718} C_DIS
LIN {X 38.9641,Y -117.445,Z 137,A -74.776,B 24.9613,C -1.4382,E1 25.0514,E2 881.0273} C_DIS
LIN {X 43.3308,Y -115.905,Z 137,A -72.473,B 24.9607,C -1.449,E1 25.0575,E2 878.7036} C_DIS
LIN {X 46.5998,Y -114.6303,Z 137,A -70.8204,B 24.9605,C -1.4527,E1 25.0618,E2 877.046} C_DIS
LIN {X 50.3725,Y -113.0227,Z 137,A -68.9807,B 24.9605,C -1.4527,E1 25.0665,E2 875.2108} C_DIS
LIN {X 53.4893,Y -111.5814,Z 137,A -67.4345,B 24.9605,C -1.453,E1 25.0704,E2 873.6678} C_DIS
LIN {X 56.9768,Y -109.8432,Z 137,A -65.0806,B 24.9588,C -1.4837,E1 25.0764,E2 871.2477} C_DIS
LIN {X 60.8661,Y -107.7374,Z 137,A -63.6628,B 24.9603,C -1.4556,E1 25.0797,E2 869.9006} C_DIS
LIN {X 63.6126,Y -106.139,Z 137,A -62.0656,B 24.9598,C -1.4647,E1 25.0835,E2 868.2868} C_DIS
LIN {X 67.1231,Y -103.9545,Z 137,A -59.8675,B 24.9588,C -1.4828,E1 25.0888,E2 866.0531} C_DIS
LIN {X 69.9517,Y -102.0721,Z 137,A -58.722,B 24.9598,C -1.4644,E1 25.0913,E2 864.9549} C_DIS
LIN {X 72.9475,Y -99.9538,Z 137,A -56.9278,B 24.9594,C -1.4727,E1 25.0954,E2 863.1472} C_DIS
LIN {X 75.8459,Y -97.7719,Z 137,A -55.1982,B 24.959,C -1.4789,E1 25.0993,E2 861.4093} C_DIS
LIN {X 81.7529,Y -92.8896,Z 137,A -51.6676,B 24.9586,C -1.4861,E1 25.1069,E2 857.8755} C_DIS
LIN {X 84.9545,Y -89.9704,Z 137,A -49.7143,B 24.9586,C -1.4882,E1 25.1108,E2 855.9251} C_DIS
LIN {X 88.777,Y -86.201,Z 137,A -46.9809,B 24.9574,C -1.5071,E1 25.1163,E2 853.1588} C_DIS
LIN {X 90.9874,Y -83.8646,Z 137,A -45.8573,B 24.9583,C -1.4922,E1 25.1183,E2 852.0752} C_DIS
LIN {X 93.2418,Y -81.3506,Z 137,A -44.1787,B 24.9577,C -1.5022,E1 25.1215,E2 850.3807} C_DIS
LIN {X 97.8895,Y -75.6943,Z 137,A -41.2243,B 24.9585,C -1.489,E1 25.1266,E2 847.4709} C_DIS
LIN {X 100.7075,Y -71.9024,Z 137,A -38.6613,B 24.957,C -1.5143,E1 25.1309,E2 844.8608} C_DIS
LIN {X 103.1226,Y -68.3947,Z 137,A -36.6437,B 24.9566,C -1.5222,E1 25.1341,E2 842.8344} C_DIS
LIN {X 105.422,Y -64.7932,Z 137,A -34.699,B 24.9564,C -1.5262,E1 25.137,E2 840.89} C_DIS
LIN {X 107.4436,Y -61.3826,Z 137,A -32.8214,B 24.9559,C -1.5338,E1 25.1396,E2 839.0043} C_DIS
LIN {X 109.8108,Y -57.0383,Z 137,A -30.7235,B 24.9561,C -1.5308,E1 25.1423,E2 836.9246} C_DIS
LIN {X 111.4578,Y -53.7481,Z 137,A -28.5212,B 24.9543,C -1.5617,E1 25.1451,E2 834.6611} C_DIS
LIN {X 113.1056,Y -50.1858,Z 137,A -26.9472,B 24.9547,C -1.5548,E1 25.1469,E2 833.1121} C_DIS
LIN {X 114.7835,Y -46.2196,Z 137,A -25.1935,B 24.9551,C -1.5486,E1 25.1487,E2 831.3827} C_DIS
LIN {X 116.2345,Y -42.4417,Z 137,A -23.079,B 24.954,C -1.5669,E1 25.1508,E2 829.2367} C_DIS
LIN {X 117.8204,Y -37.8141,Z 137,A -20.5123,B 24.9526,C -1.5898,E1 25.1531,E2 826.6306} C_DIS
LIN {X 119.1225,Y -33.4873,Z 137,A -19.297,B 24.9549,C -1.5512,E1 25.1539,E2 825.5133} C_DIS
LIN {X 120.1782,Y -29.4787,Z 137,A -16.6269,B 24.9523,C -1.5961,E1 25.1558,E2 822.7526} C_DIS
LIN {X 121.0821,Y -25.5157,Z 137,A -15.2932,B 24.9536,C -1.5739,E1 25.1566,E2 821.4792} C_DIS
LIN {X 121.5729,Y -23.0572,Z 137,A -14.0425,B 24.9531,C -1.5823,E1 25.1572,E2 820.2158} C_DIS
LIN {X 122.2887,Y -18.8959,Z 137,A -12.1204,B 24.9528,C -1.587,E1 25.1581,E2 818.294} C_DIS
LIN {X 122.8515,Y -14.803,Z 137,A -10.2269,B 24.9525,C -1.5923,E1 25.1588,E2 816.3992} C_DIS
LIN {X 123.2597,Y -10.9039,Z 137,A -8.4106,B 24.9521,C -1.5983,E1 25.1593,E2 814.5795} C_DIS
LIN {X 123.5101,Y -7.5421,Z 137,A -6.9002,B 24.952,C -1.6009,E1 25.1596,E2 813.072} C_DIS
LIN {X 123.6872,Y -3.6245,Z 137,A -5.0735,B 24.9516,C -1.6074,E1 25.1597,E2 811.2408} C_DIS
LIN {X 123.7423,Y 0.2605,Z 137,A -3.153,B 24.9509,C -1.6195,E1 25.1597,E2 809.3032} C_DIS
LIN {X 123.6694,Y 4.225,Z 137,A -1.3729,B 24.9507,C -1.6227,E1 25.1597,E2 807.5262} C_DIS
LIN {X 123.465,Y 8.2734,Z 137,A 0.5152,B 24.9503,C -1.6294,E1 25.1593,E2 805.6335} C_DIS
LIN {X 123.146,Y 12.1139,Z 137,A 2.1668,B 24.9503,C -1.6284,E1 25.1589,E2 803.9941} C_DIS
LIN {X 122.7103,Y 15.9311,Z 137,A 3.9298,B 24.95,C -1.6333,E1 25.1583,E2 802.2298} C_DIS
LIN {X 122.1892,Y 19.5386,Z 137,A 5.7255,B 24.9493,C -1.6443,E1 25.1575,E2 800.4189} C_DIS
LIN {X 121.5425,Y 23.216,Z 137,A 7.3342,B 24.9493,C -1.6436,E1 25.1567,E2 798.8211} C_DIS
LIN {X 119.9957,Y 30.2097,Z 137,A 10.3604,B 24.9497,C -1.6392,E1 25.1549,E2 795.823} C_DIS
LIN {X 118.3601,Y 36.0893,Z 137,A 13.8501,B 24.947,C -1.682,E1 25.1521,E2 792.2524} C_DIS
LIN {X 117.1597,Y 39.8208,Z 137,A 15.3219,B 24.9478,C -1.6698,E1 25.1509,E2 790.8176} C_DIS
LIN {X 115.9698,Y 43.1577,Z 137,A 16.884,B 24.9477,C -1.6708,E1 25.1494,E2 789.2619} C_DIS
LIN {X 114.7382,Y 46.3322,Z 137,A 18.4084,B 24.9476,C -1.6728,E1 25.1478,E2 787.7412} C_DIS
LIN {X 113.5353,Y 49.2062,Z 137,A 19.8472,B 24.9473,C -1.6768,E1 25.1462,E2 786.3007} C_DIS
LIN {X 110.9884,Y 54.709,Z 137,A 22.3092,B 24.9479,C -1.6673,E1 25.1434,E2 783.8744} C_DIS
LIN {X 109.2965,Y 58.0178,Z 137,A 24.2898,B 24.9468,C -1.6853,E1 25.1408,E2 781.8619} C_DIS
LIN {X 107.787,Y 60.7778,Z 137,A 25.8647,B 24.9461,C -1.6954,E1 25.1386,E2 780.2715} C_DIS
LIN {X 105.9651,Y 63.9013,Z 137,A 27.5454,B 24.9458,C -1.7003,E1 25.1362,E2 778.5879} C_DIS
LIN {X 103.6876,Y 67.5342,Z 137,A 29.5242,B 24.9455,C -1.7052,E1 25.1332,E2 776.6075} C_DIS
LIN {X 101.8147,Y 70.3269,Z 137,A 31.1362,B 24.9451,C -1.712,E1 25.1307,E2 774.9874} C_DIS
LIN {X 99.3105,Y 73.8199,Z 137,A 33.0315,B 24.9451,C -1.7123,E1 25.1276,E2 773.1005} C_DIS
LIN {X 96.706,Y 77.2006,Z 137,A 35.0348,B 24.9447,C -1.7185,E1 25.1241,E2 771.0919} C_DIS
LIN {X 93.9541,Y 80.5274,Z 137,A 37.0277,B 24.9444,C -1.7229,E1 25.1205,E2 769.0977} C_DIS
LIN {X 90.4555,Y 84.438,Z 137,A 39.2525,B 24.9447,C -1.7182,E1 25.1164,E2 766.8939} C_DIS
LIN {X 88.3602,Y 86.6281,Z 137,A 40.8183,B 24.9439,C -1.7294,E1 25.1133,E2 765.3083} C_DIS
LIN {X 85.2212,Y 89.7187,Z 137,A 42.8554,B 24.9437,C -1.7337,E1 25.1092,E2 763.2697} C_DIS
LIN {X 82.1134,Y 92.5709,Z 137,A 44.7986,B 24.9434,C -1.7372,E1 25.1052,E2 761.326} C_DIS
LIN {X 79.8768,Y 94.5081,Z 137,A 46.1695,B 24.9433,C -1.7399,E1 25.1023,E2 759.954} C_DIS
LIN {X 76.0212,Y 97.6361,Z 137,A 48.298,B 24.9435,C -1.7358,E1 25.0977,E2 757.8432} C_DIS
LIN {X 73.2204,Y 99.7534,Z 137,A 50.0912,B 24.9428,C -1.747,E1 25.0936,E2 756.0299} C_DIS
LIN {X 69.9033,Y 102.1053,Z 137,A 51.9671,B 24.9426,C -1.7499,E1 25.0893,E2 754.1537} C_DIS
LIN {X 66.8971,Y 104.0999,Z 137,A 53.4504,B 24.943,C -1.7434,E1 25.0859,E2 752.6907} C_DIS
LIN {X 63.7685,Y 106.0454,Z 137,A 55.7401,B 24.941,C -1.7749,E1 25.0802,E2 750.3337} C_DIS
LIN {X 60.1743,Y 108.1253,Z 137,A 57.1028,B 24.9426,C -1.7499,E1 25.0771,E2 749.034} C_DIS
LIN {X 56.8882,Y 109.8897,Z 137,A 58.8401,B 24.9424,C -1.7528,E1 25.0728,E2 747.2948} C_DIS
LIN {X 54.2215,Y 111.2288,Z 137,A 60.3411,B 24.9419,C -1.7604,E1 25.069,E2 745.7798} C_DIS
LIN {X 50.8061,Y 112.8288,Z 137,A 62.0166,B 24.942,C -1.759,E1 25.0647,E2 744.1118} C_DIS
LIN {X 47.7131,Y 114.1708,Z 137,A 63.5524,B 24.942,C -1.7595,E1 25.0608,E2 742.5785} C_DIS
LIN {X 44.4347,Y 115.487,Z 137,A 65.2934,B 24.9415,C -1.7663,E1 25.0562,E2 740.8252} C_DIS
LIN {X 40.6419,Y 116.875,Z 137,A 67.0551,B 24.9418,C -1.7627,E1 25.0516,E2 739.0755} C_DIS
LIN {X 37.3647,Y 117.964,Z 137,A 68.7356,B 24.9414,C -1.768,E1 25.0472,E2 737.3858} C_DIS
LIN {X 29.8077,Y 120.0978,Z 137,A 72.217,B 24.9418,C -1.7629,E1 25.0378,E2 733.9221} C_DIS
LIN {X 24.5706,Y 121.276,Z 137,A 74.5366,B 24.9422,C -1.7562,E1 25.0316,E2 731.6214} C_DIS
LIN {X 21.0429,Y 121.939,Z 137,A 76.3243,B 24.9418,C -1.7628,E1 25.0266,E2 729.8199} C_DIS
LIN {X 17.9228,Y 122.4358,Z 137,A 77.9289,B 24.9413,C -1.7701,E1 25.0221,E2 728.1997} C_DIS
LIN {X 14.4092,Y 122.8984,Z 137,A 79.5807,B 24.9413,C -1.7709,E1 25.0176,E2 726.5471} C_DIS
LIN {X 10.5007,Y 123.2937,Z 137,A 81.3444,B 24.9413,C -1.7685,E1 25.0127,E2 724.7903} C_DIS
LIN {X 7.3412,Y 123.5224,Z 137,A 82.8264,B 24.9413,C -1.7692,E1 25.0085,E2 723.3071} C_DIS
LIN {X 3.4314,Y 123.6926,Z 137,A 84.6432,B 24.9413,C -1.7693,E1 25.0035,E2 721.4907} C_DIS
LIN {X -0.4381,Y 123.7397,Z 137,A 86.4197,B 24.9413,C -1.7683,E1 24.9985,E2 719.7167} C_DIS
LIN {X -4.2635,Y 123.6679,Z 137,A 88.2711,B 24.9412,C -1.7715,E1 24.9933,E2 717.8574} C_DIS
LIN {X -7.8077,Y 123.4937,Z 137,A 89.895,B 24.9412,C -1.77,E1 24.9888,E2 716.2366} C_DIS
LIN {X -11.7849,Y 123.1776,Z 137,A 91.6993,B 24.9415,C -1.7671,E1 24.9838,E2 714.4384} C_DIS
LIN {X -15.8078,Y 122.7264,Z 137,A 93.5858,B 24.9415,C -1.7665,E1 24.9786,E2 712.5519} C_DIS
LIN {X -19.6679,Y 122.1689,Z 137,A 95.3027,B 24.9419,C -1.7611,E1 24.9739,E2 710.8464} C_DIS
LIN {X -22.941,Y 121.5951,Z 137,A 97.7103,B 24.9392,C -1.8007,E1 24.967,E2 708.3421} C_DIS
LIN {X -28.4326,Y 120.4304,Z 137,A 100.1168,B 24.94,C -1.7892,E1 24.9605,E2 705.9598} C_DIS
LIN {X -32.8806,Y 119.2922,Z 137,A 101.4777,B 24.9425,C -1.7513,E1 24.9571,E2 704.6869} C_DIS
LIN {X -36.8924,Y 118.1143,Z 137,A 103.5377,B 24.9423,C -1.7548,E1 24.9515,E2 702.6151} C_DIS
LIN {X -41.8364,Y 116.4528,Z 137,A 106.0201,B 24.9423,C -1.7549,E1 24.945,E2 700.1277} C_DIS
LIN {X -45.1538,Y 115.2075,Z 137,A 107.6526,B 24.9425,C -1.7523,E1 24.9407,E2 698.4979} C_DIS
LIN {X -48.5278,Y 113.8285,Z 137,A 109.3846,B 24.9425,C -1.7519,E1 24.9363,E2 696.7629} C_DIS
LIN {X -54.9457,Y 110.8715,Z 137,A 112.648,B 24.9428,C -1.7463,E1 24.928,E2 693.5045} C_DIS
LIN {X -58.4846,Y 109.0482,Z 137,A 114.5577,B 24.9428,C -1.7462,E1 24.9233,E2 691.5898} C_DIS
LIN {X -63.4631,Y 106.2281,Z 137,A 117.09,B 24.9435,C -1.736,E1 24.9172,E2 689.0742} C_DIS
LIN {X -66.5308,Y 104.3343,Z 137,A 118.9084,B 24.9433,C -1.7396,E1 24.9129,E2 687.2415} C_DIS
LIN {X -70.2091,Y 101.8955,Z 137,A 120.9743,B 24.9435,C -1.7366,E1 24.9081,E2 685.1759} C_DIS
LIN {X -73.5001,Y 99.5479,Z 137,A 122.771,B 24.944,C -1.7293,E1 24.9041,E2 683.3903} C_DIS
LIN {X -76.7364,Y 97.0753,Z 137,A 124.7643,B 24.944,C -1.73,E1 24.8996,E2 681.3879} C_DIS
LIN {X -80.1223,Y 94.2993,Z 137,A 126.7612,B 24.9443,C -1.7241,E1 24.8954,E2 679.3975} C_DIS
LIN {X -83.4444,Y 91.3736,Z 137,A 128.869,B 24.9444,C -1.7219,E1 24.891,E2 677.2865} C_DIS
LIN {X -86.6839,Y 88.3055,Z 137,A 130.8922,B 24.9449,C -1.715,E1 24.8869,E2 675.2713} C_DIS
LIN {X -89.7497,Y 85.1885,Z 137,A 132.9737,B 24.945,C -1.7125,E1 24.8829,E2 673.1868} C_DIS
LIN {X -92.7391,Y 81.9232,Z 137,A 134.9811,B 24.9455,C -1.7053,E1 24.8792,E2 671.1875} C_DIS
LIN {X -95.4043,Y 78.8035,Z 137,A 136.8976,B 24.9458,C -1.7011,E1 24.8757,E2 669.2724} C_DIS
LIN {X -98.0686,Y 75.4627,Z 137,A 138.9323,B 24.946,C -1.6982,E1 24.8722,E2 667.2348} C_DIS
LIN {X -100.7075,Y 71.9024,Z 137,A 140.9876,B 24.9463,C -1.6927,E1 24.8689,E2 665.1828} C_DIS
LIN {X -103.3473,Y 68.0535,Z 137,A 142.9018,B 24.9474,C -1.6756,E1 24.8659,E2 663.2998} C_DIS
LIN {X -105.0509,Y 65.3931,Z 137,A 145.025,B 24.9458,C -1.7009,E1 24.8627,E2 661.1056} C_DIS
LIN {X -107.1659,Y 61.8659,Z 137,A 146.5444,B 24.9472,C -1.678,E1 24.8606,E2 659.6326} C_DIS
LIN {X -109.9481,Y 56.7752,Z 137,A 149.0816,B 24.9482,C -1.6634,E1 24.8573,E2 657.1169} C_DIS
LIN {X -111.7441,Y 53.1489,Z 137,A 151.6098,B 24.9467,C -1.6869,E1 24.8541,E2 654.5189} C_DIS
LIN {X -113.5983,Y 49.0605,Z 137,A 152.7391,B 24.9497,C -1.6383,E1 24.853,E2 653.4993} C_DIS
LIN {X -115.5705,Y 44.22,Z 137,A 155.4972,B 24.9493,C -1.6455,E1 24.8501,E2 650.7085} C_DIS
LIN {X -116.6545,Y 41.277,Z 137,A 157.1441,B 24.949,C -1.6496,E1 24.8485,E2 649.0426} C_DIS
LIN {X -118.2777,Y 36.3587,Z 137,A 159.3768,B 24.9499,C -1.6346,E1 24.8466,E2 646.8328} C_DIS
LIN {X -119.1731,Y 33.3062,Z 137,A 160.9097,B 24.9501,C -1.6326,E1 24.8454,E2 645.296} C_DIS
LIN {X -120.0965,Y 29.8125,Z 137,A 162.6033,B 24.9503,C -1.628,E1 24.8442,E2 643.6032} C_DIS
LIN {X -121.7372,Y 22.1757,Z 137,A 166.0452,B 24.9515,C -1.6085,E1 24.8423,E2 640.1877} C_DIS
LIN {X -122.1868,Y 19.5541,Z 137,A 168.2541,B 24.9491,C -1.6479,E1 24.8413,E2 637.8716} C_DIS
LIN {X -122.9169,Y 14.2544,Z 137,A 170.5803,B 24.95,C -1.633,E1 24.8405,E2 635.567} C_DIS
LIN {X -123.3622,Y 9.6744,Z 137,A 172.229,B 24.9518,C -1.6045,E1 24.8402,E2 633.9764} C_DIS
LIN {X -123.6735,Y 4.0553,Z 137,A 174.9477,B 24.952,C -1.601,E1 24.8398,E2 631.2497} C_DIS
Enddeposition()
END
